	  "dbtags_Sterowanie".Zbiorniki_Godziny.Stop_napełnianie.HOUR := "dbHoldRegSlave_to_MT101".instHourStop_Filling;
	  "dbtags_Sterowanie".Zbiorniki_Godziny.Stop_napełnianie.MINUTE := "dbHoldRegSlave_to_MT101".instMinutStopt_Filling;
	  "dbtags_Sterowanie".Zbiorniki_Godziny.Stop_napełnianie.SECOND := 0;
	  
	  "dbtags_Sterowanie".Zbiorniki_Godziny.Start_przetłaczanie_1.HOUR := "dbHoldRegSlave_to_MT101".instHourStart_City;
	  "dbtags_Sterowanie".Zbiorniki_Godziny.Start_przetłaczanie_1.MINUTE := "dbHoldRegSlave_to_MT101".instMinutStart_City;
	  "dbtags_Sterowanie".Zbiorniki_Godziny.Start_przetłaczanie_1.SECOND := 0;
	  
	  "dbtags_Sterowanie".Zbiorniki_Godziny.Stop_przetłaczanie_1.HOUR := "dbHoldRegSlave_to_MT101".instHourStop_City;
	  "dbtags_Sterowanie".Zbiorniki_Godziny.Stop_przetłaczanie_1.MINUTE := "dbHoldRegSlave_to_MT101".instMinutStopt_City;
	  "dbtags_Sterowanie".Zbiorniki_Godziny.Stop_przetłaczanie_1.SECOND := 0;
	  
	  "dbtags_Sterowanie".Zbiorniki_Godziny.Start_dosilanie_1.HOUR := "dbHoldRegSlave_to_MT101".instHourStart_Replen;
	  "dbtags_Sterowanie".Zbiorniki_Godziny.Start_dosilanie_1.MINUTE := "dbHoldRegSlave_to_MT101".instMinutStart_Replen;
	  "dbtags_Sterowanie".Zbiorniki_Godziny.Start_dosilanie_1.SECOND := 0;
	  
	  "dbtags_Sterowanie".Zbiorniki_Godziny.Stop_dosilanie_1.HOUR := "dbHoldRegSlave_to_MT101".instHourStop_Replen;
	  "dbtags_Sterowanie".Zbiorniki_Godziny.Stop_dosilanie_1.MINUTE := "dbHoldRegSlave_to_MT101".instMinutStopt_Replen;
	  "dbtags_Sterowanie".Zbiorniki_Godziny.Stop_dosilanie_1.SECOND := 0;
	  
	  
	  
	  
	END_REGION
	
	
	
END_FUNCTION_BLOCK

FUNCTION "Zmienne_SCADA" : Void
{ S7_Optimized_Access := 'TRUE' }
VERSION : 0.1
   VAR_TEMP 
      TimeHz_DInt : DInt;
      TimeK1_ONDInt : DInt;
      TimeK2_ONDInt : DInt;
      TimeK1_OFFDInt : DInt;
      TimeK2_OFFDInt : DInt;
      tmpTimerSet_O2_Up : DInt;   // Pomocnicza wynik po mnozeniu [ms] czasu do zwiekszenia bar
      tmpQ1 : Int;   // pompcnicza przy konwersji z real do int
      tmpQ2 : Int;   // pompcnicza przy konwersji z real do int
   END_VAR


BEGIN
	(*
	//=============================================================================
	//(JZWiK S.A Radosław Tecmer)
	//(c)Copyright (2021) All Rights Reserved
	//-----------------------------------------------------------------------------
	//Testowane z:   (system docelowy z  FW 4.2)
	//Pakiet inżynierski:   TIA Portal (V14 Sp1 Update 9)
	//Ograniczenia:  ( - )
	//Wymagania:  (minimalne S7-1200 CPU 1214 FW 3.2 .)
	//Funkcjonalnośc: (Kopiowanie bloków danych z - do bloku SCADA )
	//-----------------------------------------------------------------------------
	//Zmainy wprowadzone:
	//Wersja  Data       Osoba wprowadzająca zmiany - ekspert
	//01.00.00 17.11.2021 (Tecmer Radosław - twórca) Pieresza wersja 01.00.00
	//=============================================================================
	*)
	
	//
	// Staus napędów P1 P2 P3 P4 POSTÓJ, FALOWNIK, SIEĆ
	//P1
	REGION Status napędów
	IF "IsRunInverter_P1" THEN
	  // Przekazanie wartości do instancji DB10 (1= falownik)
	  "db10organizacyjna".ins_ModeWorkContactronP1 := 1;
	  ;
	END_IF;
	IF "IsRunNetwork_P1" THEN
	  // Przekazanie wartości do instancji DB10 (2= sieć)
	  "db10organizacyjna".ins_ModeWorkContactronP1 := 2;
	  ;
	END_IF;
	IF ("IsRunNetwork_P1" = FALSE) AND ("IsRunInverter_P1" = FALSE) THEN
	  // Przekazanie wartości do instancji DB10 (0= postój)
	  "db10organizacyjna".ins_ModeWorkContactronP1 := 0;
	  ;
	END_IF;
	// P2
	IF "IsRunInverter_P2" THEN
	  // Przekazanie wartości do instancji DB10 (1= falownik)
	  "db10organizacyjna".ins_ModeWorkContactronP2 := 1;
	  ;
	END_IF;
	IF "IsRunNetwork_P2" THEN
	  // Przekazanie wartości do instancji DB10 (2= sieć)
	  "db10organizacyjna".ins_ModeWorkContactronP2 := 2;
	  ;
	END_IF;
	IF ("IsRunNetwork_P2" = FALSE) AND ("IsRunInverter_P2" = FALSE) THEN
	  // Przekazanie wartości do instancji DB10 (0= postój)
	  "db10organizacyjna".ins_ModeWorkContactronP2 := 0;
	  ;
	END_IF;
	//P3
	IF "IsRunInverter_P3" THEN
	  // Przekazanie wartości do instancji DB10 (1= falownik)
	  "db10organizacyjna".ins_ModeWorkContactronP3 := 1;
	  ;
	END_IF;
	IF "IsRunNetwork_P3" THEN
	  // Przekazanie wartości do instancji DB10 (2= sieć)
	  "db10organizacyjna".ins_ModeWorkContactronP3 := 2;
	  ;
	END_IF;
	IF ("IsRunNetwork_P3" = FALSE) AND ("IsRunInverter_P3" = FALSE) THEN
	  // Przekazanie wartości do instancji DB10 (0= postój)
	  "db10organizacyjna".ins_ModeWorkContactronP3 := 0;
	  ;
	END_IF;
	
	//P4
	IF "IsRunInverter_P4" THEN
	  // Przekazanie wartości do instancji DB10 (1= falownik)
	  "db10organizacyjna".ins_ModeWorkContactronP4 := 1;
	  ;
	END_IF;
	IF "IsRunNetwork_P4" THEN
	  // Przekazanie wartości do instancji DB10 (2= sieć)
	  "db10organizacyjna".ins_ModeWorkContactronP4 := 2;
	  ;
	END_IF;
	IF ("IsRunNetwork_P4" = FALSE) AND ("IsRunInverter_P4" = FALSE) THEN
	  // Przekazanie wartości do instancji DB10 (0= postój)
	  "db10organizacyjna".ins_ModeWorkContactronP4 := 0;
	  ;
	END_IF;
	
	//Zmienne na potrzreby trendów WinCC - Praca pomp
	//pompa P1
	IF ("IsRun_P1") = TRUE
	  
	THEN
	  "db10organizacyjna".act_stanP1 := 5;
	ELSE
	  "db10organizacyjna".act_stanP1 := 0;
	END_IF;
	//pompa P2
	IF ("IsRun_P2") = TRUE
	  
	THEN
	  "db10organizacyjna".act_statnP2 := 6;
	ELSE
	  "db10organizacyjna".act_statnP2 := 0;
	END_IF;
	//pompa P3
	IF ("IsRun_P3") = TRUE
	  
	THEN
	  "db10organizacyjna".act_stanP3 := 7;
	ELSE
	  "db10organizacyjna".act_stanP3 := 0;
	END_IF;
	
	//pompa P4
	IF ("IsRun_P3") = TRUE
	  
	THEN
	  "db10organizacyjna".act_stanP4 := 9;
	ELSE
	  "db10organizacyjna".act_stanP4 := 0;
	END_IF;
	
	
	// Zasuwy Pompownia
	// 
	// Status napędów Z11, 
	"dbdane".Z11_Status := "dbHoldRegSlave_to_MT101".instvValveZ11;
	// Status napędów Z12, 
	"dbdane".Z12_Status := "dbHoldRegSlave_to_MT101".instvValveZ12;
	
	// Staus napędów Z11 Z12
	"dbtags_Sterowanie".SetupControlPompownia.Z11_Status := "dbdane".Z11_Status;
	"dbtags_Sterowanie".SetupControlPompownia.Z12_Status := "dbdane".Z12_Status;
	
	END_REGION
	
	
	//********************
	
	
	REGION Region PID Zmienne
	  // Zmienne PID
	  //Limit górny wartości procesowej MV [%]
	  "dbdane"."PID_Compact_1_sPid_Cmpt.r_Lmn_Hlm" := "dbtags_Sterowanie".SetupControlPompownia.r_Lmn_Hlm;
	  "PID_Compact_1".sPid_Cmpt.r_Lmn_Hlm := "dbdane"."PID_Compact_1_sPid_Cmpt.r_Lmn_Hlm";
	  //Limit dolny wartości procesowej MV [%]
	  "dbdane"."PID_Compact_1_sPid_Cmpt.r_Lmn_Llm" := "dbtags_Sterowanie".SetupControlPompownia.r_Lmn_Llm;
	  "PID_Compact_1".sPid_Cmpt.r_Lmn_Llm := "dbdane"."PID_Compact_1_sPid_Cmpt.r_Lmn_Llm";
	  //Obiekt zreczywisty***
	  // Max wartość procesowa 
	  "dbdane"."PID_Compact_1sPid_Cmpt.r_Pv_Norm_OUT_2" := "dbtags_Sterowanie".SetupControlPompownia.r_Pv_Norm_OUT_2;
	  "PID_Compact_1".sPid_Cmpt.r_Pv_Norm_OUT_2 := "dbdane"."PID_Compact_1sPid_Cmpt.r_Pv_Norm_OUT_2";
	  //Min wartość procesowa
	  "dbdane"."PID_Compact_1_sPid_Cmpt.r_Pv_Norm_OUT_1" := "dbtags_Sterowanie".SetupControlPompownia.r_Pv_Norm_OUT_1;
	  "PID_Compact_1".sPid_Cmpt.r_Pv_Norm_OUT_1 := "dbdane"."PID_Compact_1_sPid_Cmpt.r_Pv_Norm_OUT_1";
	  //******
	  
	  
	  //Limmit górny zadawania
	  "dbdane"."PID_Compact_1_sPid_Cmpt.r_Sp_Hlm" := "dbtags_Sterowanie".SetupControlPompownia.r_Sp_Hlm;
	  "PID_Compact_1".sPid_Cmpt.r_Sp_Hlm := "dbdane"."PID_Compact_1_sPid_Cmpt.r_Sp_Hlm";
	  //Limit dolny zadawania
	  "dbdane"."PID_Compact_1_sPid_Cmpt.r_Sp_Llm" := "dbtags_Sterowanie".SetupControlPompownia.r_Sp_Llm;
	  "PID_Compact_1".sPid_Cmpt.r_Sp_Llm := "dbdane"."PID_Compact_1_sPid_Cmpt.r_Sp_Llm";
	  
	  // Setpoint SV
	  "db10organizacyjna".setpoint_SV_bar := "dbdane".Setpoint_SV;
	  
	END_REGION
	
	REGION Sterowanie czasem zmiany wartości ciśnienia w modelu regulacji nadążnej 
	  
	  //Opóznienie zwiększania watrości ciśnieniea  konwersja i przekaznie do zmiennej tymczasowej 
	  #tmpTimerSet_O2_Up := INT_TO_DINT("db10organizacyjna".TimeHistere_set_bar);
	  
	  //Przekazanie do Timera -Zadany czas [ms] zwłoki zwiekszenia ciśnienia
	  "dbtags_Sterowanie".SetupControlPompownia.TimerSet_O2_Up.PT := DINT_TO_TIME(#tmpTimerSet_O2_Up * "MS_TO_M");
	  //Przekazanie do Timera -Zadany czas [ms] zwłoki zmniejszenia ciśnienie
	  "dbtags_Sterowanie".SetupControlPompownia.TimerSet_O2_Down.PT := DINT_TO_TIME(#tmpTimerSet_O2_Up * "MS_TO_M");
	  
	END_REGION
	
	REGION Timery dołączenia dodatkowych pomp 
	  //***Czasy dołącz wyłacz pompy dodatkowa i oczekiwanie na Hz50 ***//
	  
	  "dbtags_Sterowanie".SetupControlPompownia.Time_ONK1 := "db10organizacyjna".Time_ONK1;
	  "dbtags_Sterowanie".SetupControlPompownia.Time_ONK2 := "db10organizacyjna".Time_ONK2;
	  "dbtags_Sterowanie".SetupControlPompownia.Time_OFFK1 := "db10organizacyjna".Time_OFFK1;
	  "dbtags_Sterowanie".SetupControlPompownia.Time_OFFK2 := "db10organizacyjna".Time_OFFK2;
	  "dbtags_Sterowanie".SetupControlPompownia.TimeHz := "db10organizacyjna".TimeHz;
	  
	  
	END_REGION
	
	
	//**
	"dbtags_Sterowanie".SetupControlPompownia.tagsdbSwitch_ModelSterowania := "dbdane".Switch_model_control_P1P4;
	
	
	
	REGION Przekazanie zmiennych sterowania
	  
	  //Wspólczynnik korekty ostrzeżęń wyokiego i niskiego PV HWrn, PV LWrn 
	  //Wsółcynnik ten koryguje poziom alarmu PID górnego i dolnego odpowiadających
	  //za dołączenie i odączenie dodatkowych kompresorów 
	  "dbtags_Sterowanie".SetupControlPompownia.PV_HWrn_correction := "db10organizacyjna".PV_HWrn_set_correct;
	  "dbtags_Sterowanie".SetupControlPompownia.PV_LWrn_correction := "db10organizacyjna".PV_LWrn_set_correct;
	  
	  //Czas oczekiwania na 50 Hz  konwersja i przekaznie do zmiennej tymczasowej 
	  #TimeHz_DInt := INT_TO_DINT("db10organizacyjna".TimeHz);
	  
	  //Czas oczekiwania na 50Hz 
	  "dbdane".TMR_Hz := DINT_TO_TIME(#TimeHz_DInt * "MS_TO_S");
	  
	  //Czas oczekiwania na K1_ON  konwersja i przekaznie do zmiennej tymczasowej 
	  #TimeK1_ONDInt := INT_TO_DINT("db10organizacyjna".Time_ONK1);
	  
	  //Czas oczekiwania na K1_ON 
	  "dbdane".TMR_ON_K1 := DINT_TO_TIME(#TimeK1_ONDInt * "MS_TO_S");
	  
	  //Czas oczekiwania na K1_OFF  konwersja i przekaznie do zmiennej tymczasowej 
	  #TimeK1_OFFDInt := INT_TO_DINT("db10organizacyjna".Time_OFFK1);
	  
	  //Czas oczekiwania na K1_OFF 
	  "dbdane".TMR_OFF_K1 := DINT_TO_TIME(#TimeK1_OFFDInt * "MS_TO_S");
	  
	  //Czas oczekiwania na K2_ON  konwersja i przekaznie do zmiennej tymczasowej 
	  #TimeK2_ONDInt := INT_TO_DINT("db10organizacyjna".Time_ONK2);
	  
	  //Czas oczekiwania na K2_ON 
	  "dbdane".TMR_ON_K2 := DINT_TO_TIME(#TimeK2_ONDInt * "MS_TO_S");
	  
	  //Czas oczekiwania na K2_OFF  konwersja i przekaznie do zmiennej tymczasowej 
	  #TimeK2_OFFDInt := INT_TO_DINT("db10organizacyjna".Time_OFFK2);
	  
	  //Czas oczekiwania na K2_OFF 
	  "dbdane".TMR_OFF_K2 := DINT_TO_TIME(#TimeK2_OFFDInt * "MS_TO_S");
	  
	  //Aktualne Hz przekazane do instancji SCADA
	  "db10organizacyjna".set_Hz_P1P4 := "dbdane".OUT_PURE_Real;
	  
	  //Aktualna zadana wartość ciśnienia do regulatora
	  CASE "dbHoldRegSlave_to_MT101".instSygSter_1 OF
	    1:
	      "dbdane".Setpoint_SV := "dbHoldRegSlave_to_MT101".instSetbarDN500_B5;
	    2:
	      "dbdane".Setpoint_SV := "dbHoldRegSlave_to_MT101".instSetbarDN225_B6;
	    3:
	      "dbdane".Setpoint_SV := "dbdane".Setpoint_bar_automat;
	      
	    ELSE
	      "dbdane".Setpoint_SV := 0.0;
	      ;
	  END_CASE;
	  
	END_REGION
	
	
	REGION Analogi 
	  
	//************ parametry analogowe**************
	//Przekazane z PLC - Zasuwy
	  "dbdane".Act_Value_B5_magistrala_bar := "dbHold_RRG".actB5_bar_magistrala;
	
	//Aktualna mierzona wartość ciśnienia zasilania B5
	"db10organizacyjna".instB5_bar_act_magistrala := "dbdane".Act_Value_B5_magistrala_bar;
	
	//Aktualna mierzona wartość ciśnienia  kierunek miasto B6
	"db10organizacyjna".instB6_bar_act_miasto := "dbdane".act_Value_B6;
	
	//Aktualna mierzona wartość ciśnienia  pompownia B7
	"db10organizacyjna".instB7_bar_act_pompownia := "dbdane".act_Value_B7;
	
	//Aktualna średnia wyliczona wartość ciśnienia 
	//Wyliczanie następuje dopiero po wybraniu sterowania od wartości średniej
	"db10organizacyjna".avg_bar:= "dbdane".actPrzepływQ1_IA_real;
	
	// Aktualne ciśnienie suchobiegu
	"db10organizacyjna".instB8_bar_act_suchobieg := "dbdane".act_Value_B8;
	END_REGION
	
	//Przekazanie zmiennej tryb pracy PID - SYMULACJA TESTY
	//IF "Sumul_OnOFF_manual_PID" = FALSE THEN
	  // ustaw trzb PID na automat
	//  "PID_Compact_1".sRet.i_Mode := "dbtags_Sterowanie".PID_Compact.Mode;
	//  ;
	//END_IF;
	
	
	REGION Alarmy 
	  // Sygnały alarmów systemu sterowania i komunikacji
	  "HMI.alarm_02" := "dbzarządzanie".sterowanie_1."alarm-warning";
	  "HMI.alarm_01" := "dbzarządzanie".sterowanie_1."alarm-modbus";
	  
	  
	END_REGION
	
	
	//Przekazanie bitu kasowania Alarmu PIEZO
	//...........
	
	
	// Falownik i zasilania RS
	REGION Counter Event OverTemp's OverVolt's from Inverters
	  // Falownik pomp
	  "db10organizacyjna".CounterOverTempFa := "dbMasterData".data26_Inver_OverTemp_415040_Fal.typeDataInverter_int[0];
	  "db10organizacyjna".CounterOverVoltFal := "dbMasterData".data26_Inver_OverVolts_415050_Fal.typeDataInverter_int[0];
	  "HMI.gotowość_falownik_1" := "dbzarządzanie".awaria_falownika_F1;
	  // RS
	  "HMI.brak_zasilania" := "dbzarządzanie".brak_zasilania_RS;
	  
	
	END_REGION
	
	
	REGION Manual zadane Hz (SV)
	  // konwertowanie wartości manualnie zadawanych Hz z Real do Word
	  "dbdane".tmpManualSV := REAL_TO_LREAL("dbdane".Manual_SV);
	  "dbdane".ManualSV_Int := LREAL_TO_INT( "dbdane".tmpManualSV);
	 
	  
	END_REGION
	
	
	
	REGION Modbus staus, error
	  // Status Modbus slave
	  "db10organizacyjna".RTU_MPP04_1errorStatus := "dbTags_master_MPP04_1".modbusMaster.errorStatus;
	  "db10organizacyjna".RTU_MPP04_2errorStatus := "dbTags_master_MPP04_2".modbusMaster.errorStatus;
	  "db10organizacyjna".RTU_Fal_1errorStatus := "dbTags_master_Fal_1".modbusMaster.errorStatus;
	  //Status Modbus master
	  "db10organizacyjna".RTU_MT101 := "dbTags_slave_RTU".modbusMaster.errorStatus;
	  %DB10.DBX25.0 := "dbzarządzanie".sterowanie_1.awaria_modbus_falownik;
	  %DB10.DBX25.1 := "dbzarządzanie".sterowanie_1.awaria_modbus_przepływ_pomp;
	  %DB10.DBX25.2 := "dbzarządzanie".sterowanie_1.awaria_modbus_przepływ_magist;
	  %DB10.DBX25.3 := "dbzarządzanie".sterowanie_1.awaria_modbus_mt101;
	  
	  
	END_REGION
	
	REGION Modbus master PLC S7 1200 - Przepływomierz Q1 pompownia
	  // przekazanie wartości Real
	  "db10organizacyjna".instFlowDN225_act_Q1 := "dbdane".Wielkość_przeływu_Q1;
	  
	  // konwertowanie do Int
	  "db10organizacyjna".actQ1_przepyw_pompownia_Int := "dbdane".actPrzeoływQ1;
	  
	  // Sumay przepływu 
	  "db10organizacyjna".instSumFlowDN225_Q1 := "dbdane".Licznik_objętość_VF_Q1;
	  
	  
	  //******* Dopisać jeśli potzrebne do wizualizacji 
	  // Adres 2 - Licznik_objętość_VF
	  // Adres 4- stan bierzący licznika objetości w stecz VR
	  // Adres 6- stan bierzący licznika różnicowego  objętości VD
	  // Adres 8- główny liczni objetości w przód GF
	  // Adres 10- główny liczni objetości w stecz GR
	  // Adres 12- główny lróznicowy liczni objetościGD
	  // Status MP04 Q1 - pompownia
	  
	  
	END_REGION
	
	
	REGION Modbus master PLC S7 1200 - Przepływomierz Q2 Zasuwy
	  // przekazanie wartości
	  "db10organizacyjna".instFlowDN500_act_Q2 := "dbdane".Wielkość_przeływu_Q2;
	  
	  // konwertowanie do Int
	  #tmpQ2 := REAL_TO_INT("db10organizacyjna".instFlowDN500_act_Q2);
	  "db10organizacyjna".actQ2_przepyw_pompownia_Int := #tmpQ2;
	  
	  //******* Dopisać jeśli potzrebne do wizualizacji 
	  // Adres 2 - Licznik_objętość_VF
	  // Adres 4- stan bierzący licznika objetości w stecz VR
	  // Adres 6- stan bierzący licznika różnicowego  objętości VD
	  // Adres 8- główny liczni objetości w przód GF
	  // Adres 10- główny liczni objetości w stecz GR
	  // Adres 12- główny lróznicowy liczni objetościGD
	  // Status MP04 Q1 - pompownia
	  
	  
	  
	  // Sumay przepływu 
	  "db10organizacyjna".instSumFlowDN500_Q2 := "dbdane".Licznik_objętość_VF_Q2;
	  
	END_REGION
	
	REGION Modbus RTU Falownik 
	  // Słowo statusu 
	  "HMI.SłowoStatus_Falownik1" := "dbModbusRTU_Reg".received26_Inver_Status_word_416030.typeDataInverter_int[0];
	  
	END_REGION
	
	REGION położenie Z10
	  // kopiowanie odebranych danych z PLC Zasuwy
	  "dbHoldRegSlave_to_MT101".instPozitionZ10_act := INT_TO_REAL("db10organizacyjna".actPozycja_Z10);
	  
	END_REGION
	
	
	
	
	
	
	  
	  
	
	
	
	
END_FUNCTION

FUNCTION "Konwersja_Time_to_Int" : Void
{ S7_Optimized_Access := 'TRUE' }
AUTHOR : RTecmer
FAMILY : 'HMI(XM)'
VERSION : 0.1
//Przekazywanie zmiennych między urządzeniami

BEGIN
	(*
	//=============================================================================
	//(JZWiK S.A Radosław Tecmer)
	//(c)Copyright (2021) All Rights Reserved
	//-----------------------------------------------------------------------------
	//Testowane z:   (system docelowy z  FW 4.2)
	//Pakiet inżynierski:   TIA Portal (V14 Sp1 Update 9)
	//Ograniczenia:  ( - )
	//Wymagania:  (minimalne S7-1200 CPU 1214 FW 3.2 .)
	//Funkcjonalnośc: (KOnwerja zmiennych formatu Time of Day na Int )
	//-----------------------------------------------------------------------------
	//Zmainy wprowadzone:
	//Wersja  Data       Osoba wprowadzająca zmiany - ekspert
	//01.00.00 17.02.2022 (Tecmer Radosław - twórca) Pieresza wersja 01.00.00
	//=============================================================================
	*)
	
	// Aktualny czas
	"Konverter_zegarów"(HOUR:="Data_Czas_synch".Time_Local_read.HOUR,
	                    MINUTE:="Data_Czas_synch".Time_Local_read.MINUTE,
	                    SECOND:="Data_Czas_synch".Time_Local_read.SECOND,
	                    Czas_Liczba_conv_Real=>"db10organizacyjna".actTime,
	                    Zegar_H=>"db10organizacyjna".actHour,
	                    Zegar_M=>"db10organizacyjna".actMinut,
	                    Zegar_S=>"db10organizacyjna".actSec);
	
	
	// Godzina start napełniania
	"Konverter_zegarów"(HOUR:="db10organizacyjna".instHourStart_Filling.HOUR,
	                    MINUTE:="db10organizacyjna".instHourStart_Filling.MINUTE,
	                    SECOND:="db10organizacyjna".instHourStart_Filling.SECOND,
	                    Czas_Liczba_conv_Real=>"dbzarządzanie".instHourStart_Filling,
	                    Zegar_H=>"db10organizacyjna".instHourStart_Filling_1,
	                    Zegar_M=>"db10organizacyjna".instMinutStart_Filling,
	                    Zegar_S=>"db10organizacyjna".instSecStart_Filling_1);
	
	
	// Godzina stop napełniania
	"Konverter_zegarów"(HOUR := "db10organizacyjna".instHourStop_Filling.HOUR,
	                    MINUTE := "db10organizacyjna".instHourStop_Filling.MINUTE,
	                    SECOND := "db10organizacyjna".instHourStop_Filling.SECOND,
	                    Czas_Liczba_conv_Real => "dbzarządzanie".instHourStop_Filling,
	                    Zegar_H=>"db10organizacyjna".instHourStop_Filling_1,
	                    Zegar_M=>"db10organizacyjna".instMinutStopt_Filling,
	                    Zegar_S=>"db10organizacyjna".instSecStop_Filling_1);
	
	// Godzina start przetłaczanie miasto DN225
	"Konverter_zegarów"(HOUR := "db10organizacyjna".instHourStart_City.HOUR,
	                    MINUTE := "db10organizacyjna".instHourStart_City.MINUTE,
	                    SECOND := "db10organizacyjna".instHourStart_City.SECOND,
	                    Czas_Liczba_conv_Real => "dbzarządzanie".instHourStart_City,
	                    Zegar_H=>"db10organizacyjna".instHourStart_City_1,
	                    Zegar_M=>"db10organizacyjna".instMinutStart_City,
	                    Zegar_S=>"db10organizacyjna".instSecStart_City_1);
	
	
	// Godzina stop przetłaczanie miasto DN225
	"Konverter_zegarów"(HOUR := "db10organizacyjna".instHourStop_City.HOUR,
	                    MINUTE := "db10organizacyjna".instHourStop_City.MINUTE,
	                    SECOND := "db10organizacyjna".instHourStop_City.SECOND,
	                    Czas_Liczba_conv_Real => "dbzarządzanie".instHourStop_City,
	                    Zegar_H=>"db10organizacyjna".instHourStop_City_1,
	                    Zegar_M=>"db10organizacyjna".instMinutStopt_City,
	                    Zegar_S=>"db10organizacyjna".instSecStop_City_1);
	
	
	// Godzina start dosilanie DN500
	"Konverter_zegarów"(HOUR := "db10organizacyjna".instHourStart_Replen.HOUR,
	                    MINUTE := "db10organizacyjna".instHourStart_Replen.MINUTE,
	                    SECOND := "db10organizacyjna".instHourStart_Replen.SECOND,
	                    Czas_Liczba_conv_Real => "dbzarządzanie".instHourStart_Replen,
	                    Zegar_H=>"db10organizacyjna".instHourStart_Replen_1,
	                    Zegar_M=>"db10organizacyjna".instMinutStart_Replen,
	                    Zegar_S=>"db10organizacyjna".instSecStart_Replen_1);
	
	
	
	
	
	// Godzina stop dosilanie DN500
	"Konverter_zegarów"(HOUR :="db10organizacyjna".instHourStop_Replen.HOUR,
	                    MINUTE :="db10organizacyjna".instHourStop_Replen.MINUTE,
	                    SECOND :="db10organizacyjna".instHourStop_Replen.SECOND,
	                    Czas_Liczba_conv_Real => "dbzarządzanie".instHourStop_Replen,
	                    Zegar_H=>"db10organizacyjna".instHourStop_Replen_1,
	                    Zegar_M=>"db10organizacyjna".instMinutStopt_Replen,
	                    Zegar_S=>"db10organizacyjna".instSecStop_Replen_1);
	
	
	
	
	
	
	
	
	
	
	
END_FUNCTION

FUNCTION "Konverter_zegarów" : Void   // FC31, LAD
{ S7_Optimized_Access := 'FALSE' }
VERSION : 0.1
// stored: AutoNumber true, IsIECCheckEnabled false, SetENOAutomatically false, UDAEnableTagReadback false
   VAR_INPUT
      HOUR : USInt;   // Zmienna godzina z DTL
      MINUTE : USInt;   // Zmienna minuty z DTL
      SECOND : USInt;   // Zmienne sekundy z DTL
   END_VAR
   VAR_OUTPUT
      Czas_Liczba_conv_Real : Real;   // Liczba przedstawiająca czas 00:00:00 liczbowo 00.0000
      Zegar_H : Int;
      Zegar_M : Int;
      Zegar_S : Int;
   END_VAR
   VAR_TEMP
      zegar_H_pomocnicza : Real;   // pomocnicza do przekształcenia czasu z DLT do Real
      zegar_M_pomocnicza : Real;   // pomocnicza do przekształcenia czasu z DLT do Real
      zegar_S_pomocnicza : Real;   // pomocnicza do przekształcenia czasu z DLT do Real
      zegar_H_Uint : UInt;   // pomocnicza do przekształcenia czasu z DLT do Uint
      zegar_M_Uint : UInt;   // pomocnicza do przekształcenia czasu z DLT do Uint
      zegar_S_Uint : UInt;   // pomocnicza do przekształcenia czasu z DLT do Uint
   END_VAR
BEGIN

REGION Network 1: Wyodrębnienie zegara z danej DTL czasu lokalnego
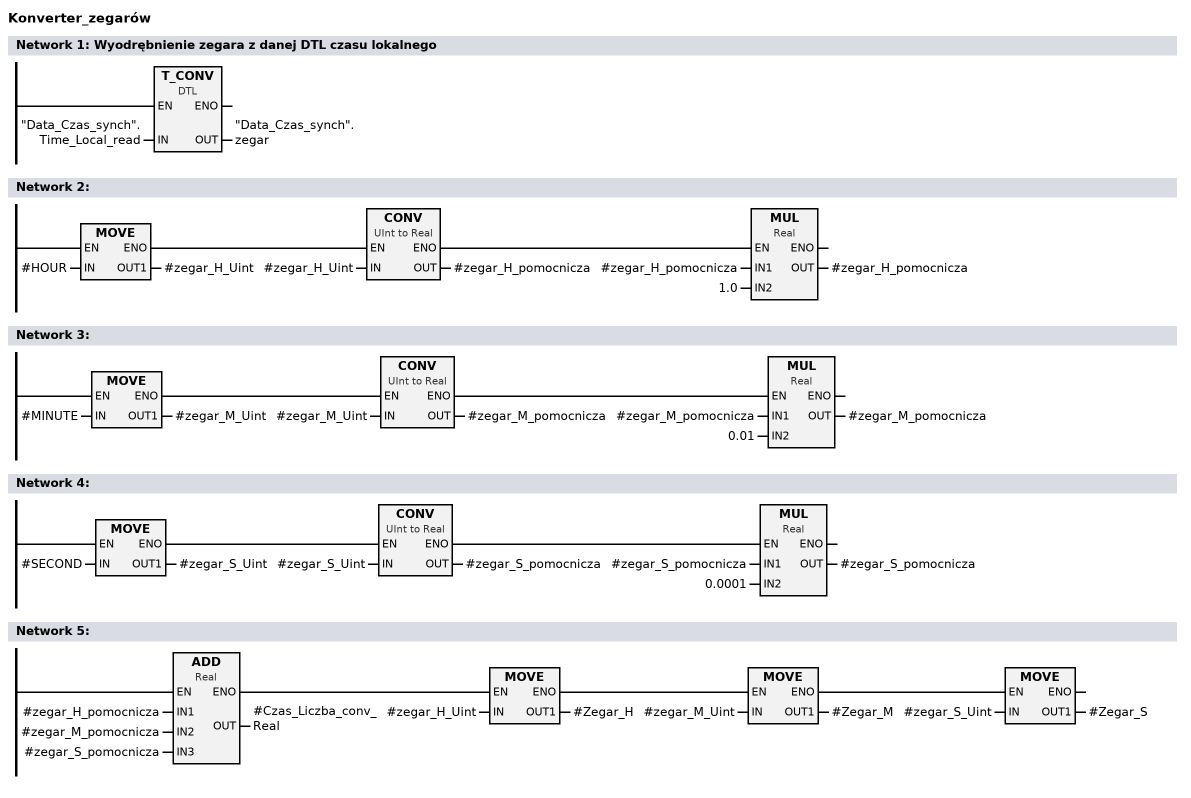
   RUNG wire#powerrail
      { S7_Templates := "[src_type := DTL, dest_type := Time_Of_Day]" } T_CONV(IN := "Data_Czas_synch".Time_Local_read, OUT => "Data_Czas_synch".zegar)
   END_RUNG
   // the same network as SCL:
   T_CONV(IN := "Data_Czas_synch".Time_Local_read, OUT => "Data_Czas_synch".zegar);
END_REGION

REGION Network 2
   RUNG wire#powerrail
      { S7_GenerateENO := "TRUE" } Move(in := #HOUR, out1 => #zegar_H_Uint)
      { S7_Templates := "[SrcType := UInt, DestType := Real]"; S7_GenerateENO := "TRUE" } Convert(in := #zegar_H_Uint, out => #zegar_H_pomocnicza)
      { S7_Templates := "SrcType := Real"; S7_GenerateENO := "TRUE" } Mul(in1 := #zegar_H_pomocnicza, in2 := 1.0, out => #zegar_H_pomocnicza)
   END_RUNG
   // the same network as SCL:
   // ENO of a box is taken as its EN; it also drops when the box reports an error
   #zegar_H_Uint := #HOUR;
   #zegar_H_pomocnicza := UINT_TO_REAL(#zegar_H_Uint);
   #zegar_H_pomocnicza := #zegar_H_pomocnicza * 1.0;
END_REGION

REGION Network 3
   RUNG wire#powerrail
      { S7_GenerateENO := "TRUE" } Move(in := #MINUTE, out1 => #zegar_M_Uint)
      { S7_Templates := "[SrcType := UInt, DestType := Real]"; S7_GenerateENO := "TRUE" } Convert(in := #zegar_M_Uint, out => #zegar_M_pomocnicza)
      { S7_Templates := "SrcType := Real"; S7_GenerateENO := "TRUE" } Mul(in1 := #zegar_M_pomocnicza, in2 := 0.01, out => #zegar_M_pomocnicza)
   END_RUNG
   // the same network as SCL:
   // ENO of a box is taken as its EN; it also drops when the box reports an error
   #zegar_M_Uint := #MINUTE;
   #zegar_M_pomocnicza := UINT_TO_REAL(#zegar_M_Uint);
   #zegar_M_pomocnicza := #zegar_M_pomocnicza * 0.01;
END_REGION

REGION Network 4
   RUNG wire#powerrail
      { S7_GenerateENO := "TRUE" } Move(in := #SECOND, out1 => #zegar_S_Uint)
      { S7_Templates := "[SrcType := UInt, DestType := Real]"; S7_GenerateENO := "TRUE" } Convert(in := #zegar_S_Uint, out => #zegar_S_pomocnicza)
      { S7_Templates := "SrcType := Real"; S7_GenerateENO := "TRUE" } Mul(in1 := #zegar_S_pomocnicza, in2 := 0.0001, out => #zegar_S_pomocnicza)
   END_RUNG
   // the same network as SCL:
   // ENO of a box is taken as its EN; it also drops when the box reports an error
   #zegar_S_Uint := #SECOND;
   #zegar_S_pomocnicza := UINT_TO_REAL(#zegar_S_Uint);
   #zegar_S_pomocnicza := #zegar_S_pomocnicza * 0.0001;
END_REGION

REGION Network 5
   RUNG wire#powerrail
      { S7_Templates := "SrcType := Real"; S7_GenerateENO := "TRUE" } Add(in1 := #zegar_H_pomocnicza, in2 := #zegar_M_pomocnicza, in3 := #zegar_S_pomocnicza, out => #Czas_Liczba_conv_Real)
      Move(in := #zegar_H_Uint, out1 => #Zegar_H)
      Move(in := #zegar_M_Uint, out1 => #Zegar_M)
      Move(in := #zegar_S_Uint, out1 => #Zegar_S)
   END_RUNG
   // the same network as SCL:
   // ENO of a box is taken as its EN; it also drops when the box reports an error
   #Czas_Liczba_conv_Real := #zegar_H_pomocnicza + #zegar_M_pomocnicza + #zegar_S_pomocnicza;
   #Zegar_H := #zegar_H_Uint;
   #Zegar_M := #zegar_M_Uint;
   #Zegar_S := #zegar_S_Uint;
END_REGION
END_FUNCTION

FUNCTION "Kontrola trybu sterowania" : Void   // FC27, LAD
{ S7_Optimized_Access := 'TRUE' }
AUTHOR : rtecmer
VERSION : 0.1
// Kontrola trybu pracy Manual/Automat. Kontrola trybu pracy PID tryb 4 / tryb 3. Sprawdzanie stanu otwarcia Z11, Z12. Sprawdzanie sygnału Alarm Suchobieg. Tryb sterownia zostaje przerwany w wypadku wystąpienia 'Suchobiegu", lub zamknięcia obu zasów Z11 i Z12
// stored: AutoNumber true, IsIECCheckEnabled false, SetENOAutomatically false, UDAEnableTagReadback false
   VAR_IN_OUT
      Timer_Reset_delay : TOF_TIME;
   END_VAR
   VAR_TEMP   // added for the SCL form of the ladder/FBD networks
      _w1 : Bool;
      _w2 : Bool;
   END_VAR
BEGIN

REGION Network 1: Ustawienie pracy [Automat]
   // Ustawienie bitu [Automat] przełacznikiem trybu pracy
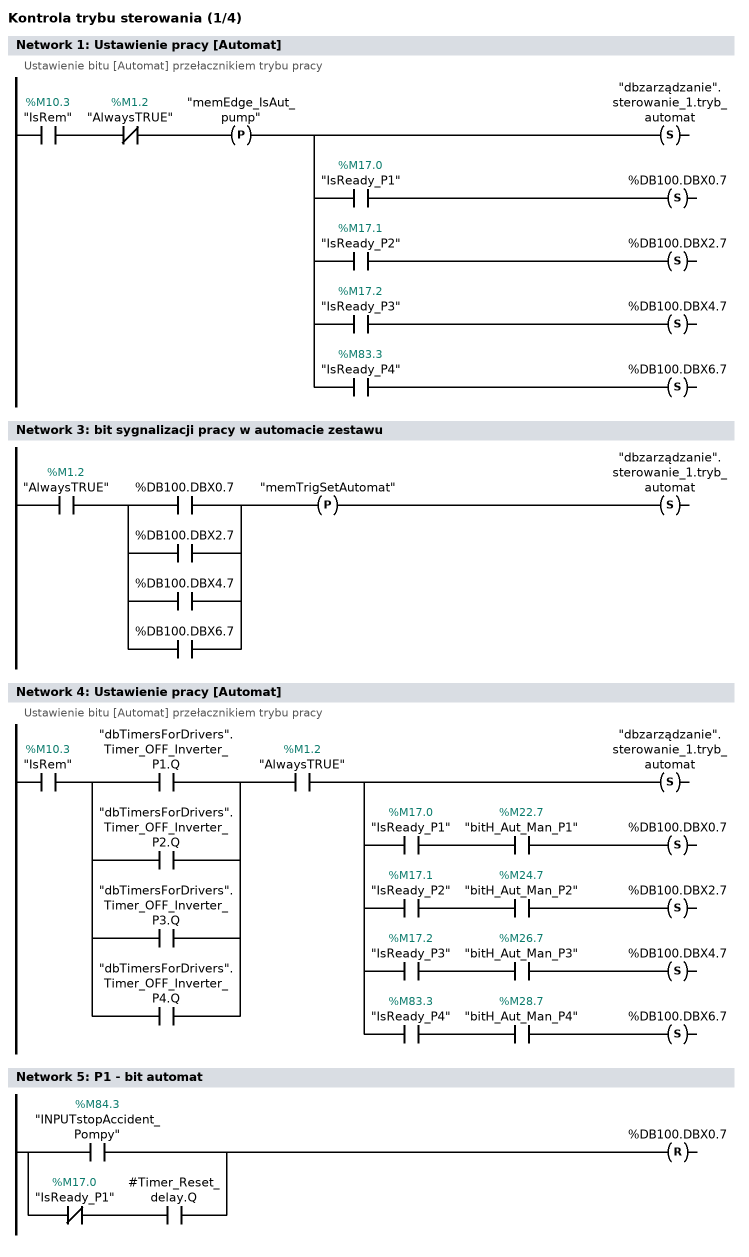
   RUNG wire#powerrail
      Contact( "IsRem" )
      I_Contact( "AlwaysTRUE" )
      P_Trig( "memEdge_IsAut_pump" )
      wire#w1
      S_Coil( "dbzarządzanie".sterowanie_1.tryb_automat )
   END_RUNG
   RUNG wire#w1
      Contact( "IsReady_P1" )
      S_Coil( %DB100.DBX0.7 )
   END_RUNG
   RUNG wire#w1
      Contact( "IsReady_P2" )
      S_Coil( %DB100.DBX2.7 )
   END_RUNG
   RUNG wire#w1
      Contact( "IsReady_P3" )
      S_Coil( %DB100.DBX4.7 )
   END_RUNG
   RUNG wire#w1
      Contact( "IsReady_P4" )
      S_Coil( %DB100.DBX6.7 )
   END_RUNG
   // the same network as SCL:
   #_w1 := "IsRem" AND NOT "AlwaysTRUE";
   #_w2 := #_w1 AND NOT "memEdge_IsAut_pump";   // rising edge
   "memEdge_IsAut_pump" := #_w1;
   IF #_w2 THEN "dbzarządzanie".sterowanie_1.tryb_automat := TRUE; END_IF;
   IF #_w2 AND "IsReady_P1" THEN %DB100.DBX0.7 := TRUE; END_IF;
   IF #_w2 AND "IsReady_P2" THEN %DB100.DBX2.7 := TRUE; END_IF;
   IF #_w2 AND "IsReady_P3" THEN %DB100.DBX4.7 := TRUE; END_IF;
   IF #_w2 AND "IsReady_P4" THEN %DB100.DBX6.7 := TRUE; END_IF;
END_REGION

REGION Network 3: bit sygnalizacji pracy w automacie zestawu
   RUNG wire#powerrail
      Contact( "AlwaysTRUE" )
      wire#w1
      Contact( %DB100.DBX0.7 )
      wire#w2
      P_Trig( "memTrigSetAutomat" )
      S_Coil( "dbzarządzanie".sterowanie_1.tryb_automat )
   END_RUNG
   RUNG wire#w1
      Contact( %DB100.DBX2.7 )
   END_RUNG wire#w2
   RUNG wire#w1
      Contact( %DB100.DBX4.7 )
   END_RUNG wire#w2
   RUNG wire#w1
      Contact( %DB100.DBX6.7 )
   END_RUNG wire#w2
   // the same network as SCL:
   #_w1 := "AlwaysTRUE" AND (%DB100.DBX0.7 OR %DB100.DBX2.7 OR %DB100.DBX4.7 OR %DB100.DBX6.7);
   #_w2 := #_w1 AND NOT "memTrigSetAutomat";   // rising edge
   "memTrigSetAutomat" := #_w1;
   IF #_w2 THEN "dbzarządzanie".sterowanie_1.tryb_automat := TRUE; END_IF;
END_REGION

REGION Network 4: Ustawienie pracy [Automat]
   // Ustawienie bitu [Automat] przełacznikiem trybu pracy
   RUNG wire#powerrail
      Contact( "IsRem" )
      wire#w1
      Contact( "dbTimersForDrivers".Timer_OFF_Inverter_P1.Q )
      wire#w2
      Contact( "AlwaysTRUE" )
      wire#w3
      S_Coil( "dbzarządzanie".sterowanie_1.tryb_automat )
   END_RUNG
   RUNG wire#w1
      Contact( "dbTimersForDrivers".Timer_OFF_Inverter_P2.Q )
   END_RUNG wire#w2
   RUNG wire#w1
      Contact( "dbTimersForDrivers".Timer_OFF_Inverter_P3.Q )
   END_RUNG wire#w2
   RUNG wire#w1
      Contact( "dbTimersForDrivers".Timer_OFF_Inverter_P4.Q )
   END_RUNG wire#w2
   RUNG wire#w3
      Contact( "IsReady_P1" )
      Contact( "bitH_Aut_Man_P1" )
      S_Coil( %DB100.DBX0.7 )
   END_RUNG
   RUNG wire#w3
      Contact( "IsReady_P2" )
      Contact( "bitH_Aut_Man_P2" )
      S_Coil( %DB100.DBX2.7 )
   END_RUNG
   RUNG wire#w3
      Contact( "IsReady_P3" )
      Contact( "bitH_Aut_Man_P3" )
      S_Coil( %DB100.DBX4.7 )
   END_RUNG
   RUNG wire#w3
      Contact( "IsReady_P4" )
      Contact( "bitH_Aut_Man_P4" )
      S_Coil( %DB100.DBX6.7 )
   END_RUNG
   // the same network as SCL:
   #_w1 := "IsRem" AND ("dbTimersForDrivers".Timer_OFF_Inverter_P1.Q OR "dbTimersForDrivers".Timer_OFF_Inverter_P2.Q OR "dbTimersForDrivers".Timer_OFF_Inverter_P3.Q OR "dbTimersForDrivers".Timer_OFF_Inverter_P4.Q) AND "AlwaysTRUE";
   IF #_w1 THEN "dbzarządzanie".sterowanie_1.tryb_automat := TRUE; END_IF;
   IF #_w1 AND "IsReady_P1" AND "bitH_Aut_Man_P1" THEN %DB100.DBX0.7 := TRUE; END_IF;
   IF #_w1 AND "IsReady_P2" AND "bitH_Aut_Man_P2" THEN %DB100.DBX2.7 := TRUE; END_IF;
   IF #_w1 AND "IsReady_P3" AND "bitH_Aut_Man_P3" THEN %DB100.DBX4.7 := TRUE; END_IF;
   IF #_w1 AND "IsReady_P4" AND "bitH_Aut_Man_P4" THEN %DB100.DBX6.7 := TRUE; END_IF;
END_REGION

REGION Network 5: P1 - bit automat
   RUNG wire#powerrail
      Contact( "INPUTstopAccident_Pompy" )
      wire#w1
      R_Coil( %DB100.DBX0.7 )
   END_RUNG
   RUNG wire#powerrail
      I_Contact( "IsReady_P1" )
      Contact( #Timer_Reset_delay.Q )
   END_RUNG wire#w1
   // the same network as SCL:
   IF "INPUTstopAccident_Pompy" OR (NOT "IsReady_P1" AND #Timer_Reset_delay.Q) THEN
       %DB100.DBX0.7 := FALSE;
   END_IF;
END_REGION

REGION Network 6: P2 - bit automat
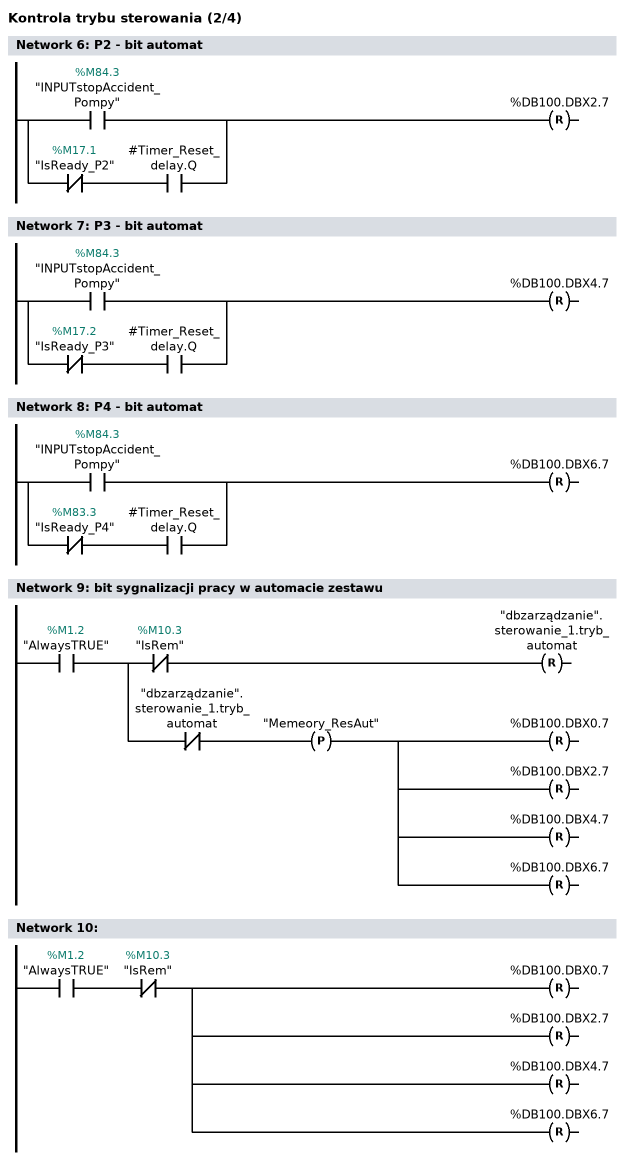
   RUNG wire#powerrail
      Contact( "INPUTstopAccident_Pompy" )
      wire#w1
      R_Coil( %DB100.DBX2.7 )
   END_RUNG
   RUNG wire#powerrail
      I_Contact( "IsReady_P2" )
      Contact( #Timer_Reset_delay.Q )
   END_RUNG wire#w1
   // the same network as SCL:
   IF "INPUTstopAccident_Pompy" OR (NOT "IsReady_P2" AND #Timer_Reset_delay.Q) THEN
       %DB100.DBX2.7 := FALSE;
   END_IF;
END_REGION

REGION Network 7: P3 - bit automat
   RUNG wire#powerrail
      Contact( "INPUTstopAccident_Pompy" )
      wire#w1
      R_Coil( %DB100.DBX4.7 )
   END_RUNG
   RUNG wire#powerrail
      I_Contact( "IsReady_P3" )
      Contact( #Timer_Reset_delay.Q )
   END_RUNG wire#w1
   // the same network as SCL:
   IF "INPUTstopAccident_Pompy" OR (NOT "IsReady_P3" AND #Timer_Reset_delay.Q) THEN
       %DB100.DBX4.7 := FALSE;
   END_IF;
END_REGION

REGION Network 8: P4 - bit automat
   RUNG wire#powerrail
      Contact( "INPUTstopAccident_Pompy" )
      wire#w1
      R_Coil( %DB100.DBX6.7 )
   END_RUNG
   RUNG wire#powerrail
      I_Contact( "IsReady_P4" )
      Contact( #Timer_Reset_delay.Q )
   END_RUNG wire#w1
   // the same network as SCL:
   IF "INPUTstopAccident_Pompy" OR (NOT "IsReady_P4" AND #Timer_Reset_delay.Q) THEN
       %DB100.DBX6.7 := FALSE;
   END_IF;
END_REGION

REGION Network 9: bit sygnalizacji pracy w automacie zestawu
   RUNG wire#powerrail
      Contact( "AlwaysTRUE" )
      wire#w1
      I_Contact( "IsRem" )
      R_Coil( "dbzarządzanie".sterowanie_1.tryb_automat )
   END_RUNG
   RUNG wire#w1
      I_Contact( "dbzarządzanie".sterowanie_1.tryb_automat )
      P_Trig( "Memeory_ResAut" )
      wire#w2
      R_Coil( %DB100.DBX0.7 )
   END_RUNG
   RUNG wire#w2
      R_Coil( %DB100.DBX2.7 )
   END_RUNG
   RUNG wire#w2
      R_Coil( %DB100.DBX4.7 )
   END_RUNG
   RUNG wire#w2
      R_Coil( %DB100.DBX6.7 )
   END_RUNG
   // the same network as SCL:
   IF "AlwaysTRUE" AND NOT "IsRem" THEN "dbzarządzanie".sterowanie_1.tryb_automat := FALSE; END_IF;
   #_w1 := "AlwaysTRUE" AND NOT "dbzarządzanie".sterowanie_1.tryb_automat;
   #_w2 := #_w1 AND NOT "Memeory_ResAut";   // rising edge
   "Memeory_ResAut" := #_w1;
   IF #_w2 THEN
       %DB100.DBX0.7 := FALSE;
       %DB100.DBX2.7 := FALSE;
       %DB100.DBX4.7 := FALSE;
       %DB100.DBX6.7 := FALSE;
   END_IF;
END_REGION

REGION Network 10
   RUNG wire#powerrail
      Contact( "AlwaysTRUE" )
      I_Contact( "IsRem" )
      wire#w1
      R_Coil( %DB100.DBX0.7 )
   END_RUNG
   RUNG wire#w1
      R_Coil( %DB100.DBX2.7 )
   END_RUNG
   RUNG wire#w1
      R_Coil( %DB100.DBX4.7 )
   END_RUNG
   RUNG wire#w1
      R_Coil( %DB100.DBX6.7 )
   END_RUNG
   // the same network as SCL:
   IF "AlwaysTRUE" AND NOT "IsRem" THEN
       %DB100.DBX0.7 := FALSE;
       %DB100.DBX2.7 := FALSE;
       %DB100.DBX4.7 := FALSE;
       %DB100.DBX6.7 := FALSE;
   END_IF;
END_REGION

REGION Network 11: PID is auto = 3 , mamual =4
   // PID tryb manualnye = ON/OFF
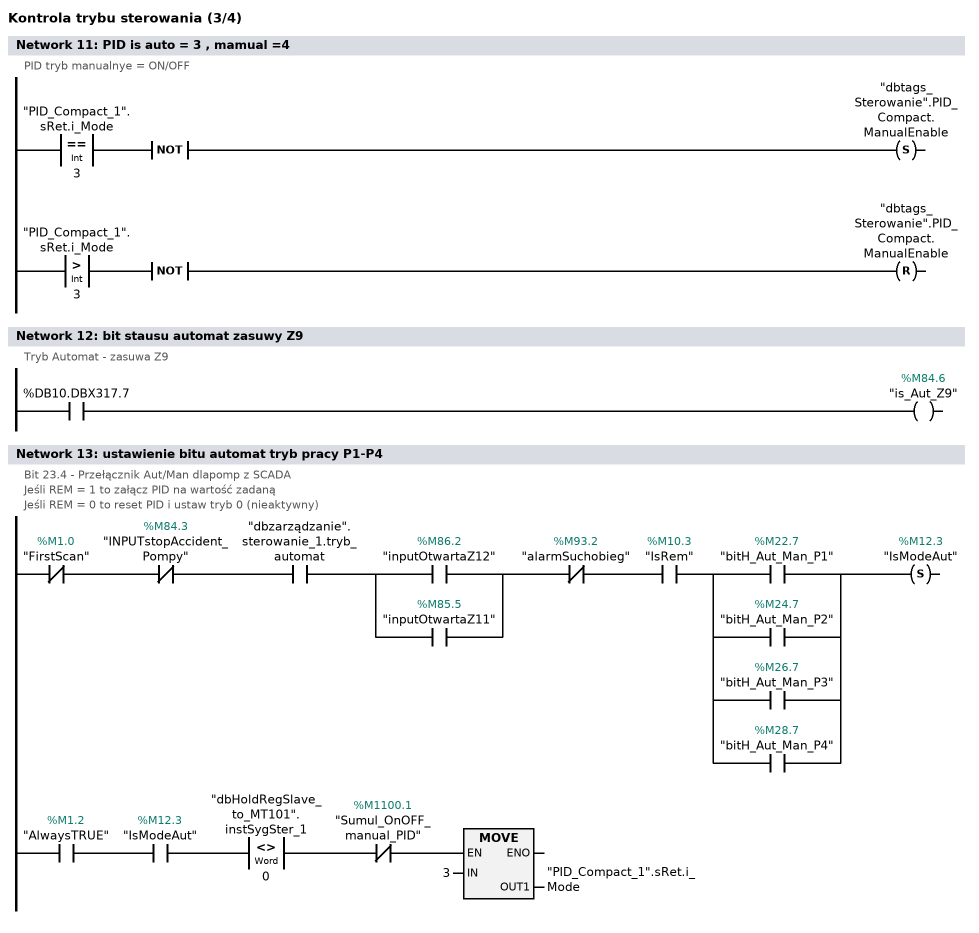
   RUNG wire#powerrail
      { S7_Templates := "SrcType := Int" } EQ_Contact(in1 := "PID_Compact_1".sRet.i_Mode, in2 := 3)
      Not()
      S_Coil( "dbtags_Sterowanie".PID_Compact.ManualEnable )
   END_RUNG
   RUNG wire#powerrail
      { S7_Templates := "SrcType := Int" } GT_Contact(in1 := "PID_Compact_1".sRet.i_Mode, in2 := 3)
      Not()
      R_Coil( "dbtags_Sterowanie".PID_Compact.ManualEnable )
   END_RUNG
   // the same network as SCL:
   IF NOT ("PID_Compact_1".sRet.i_Mode = 3) THEN
       "dbtags_Sterowanie".PID_Compact.ManualEnable := TRUE;
   END_IF;
   IF NOT ("PID_Compact_1".sRet.i_Mode > 3) THEN
       "dbtags_Sterowanie".PID_Compact.ManualEnable := FALSE;
   END_IF;
END_REGION

REGION Network 12: bit stausu automat zasuwy Z9
   // Tryb Automat - zasuwa Z9
   RUNG wire#powerrail
      Contact( %DB10.DBX317.7 )
      Coil( "is_Aut_Z9" )
   END_RUNG
   // the same network as SCL:
   "is_Aut_Z9" := %DB10.DBX317.7;
END_REGION

REGION Network 13: ustawienie bitu automat tryb pracy P1-P4
   // Bit 23.4 - Przełącznik Aut/Man dlapomp z SCADA
   // Jeśli REM = 1 to załącz PID na wartość zadaną
   // Jeśli REM = 0 to reset PID i ustaw tryb 0 (nieaktywny)
   RUNG wire#powerrail
      I_Contact( "FirstScan" )
      I_Contact( "INPUTstopAccident_Pompy" )
      Contact( "dbzarządzanie".sterowanie_1.tryb_automat )
      wire#w1
      Contact( "inputOtwartaZ12" )
      wire#w2
      I_Contact( "alarmSuchobieg" )
      Contact( "IsRem" )
      wire#w3
      Contact( "bitH_Aut_Man_P1" )
      wire#w4
      S_Coil( "IsModeAut" )
   END_RUNG
   RUNG wire#w1
      Contact( "inputOtwartaZ11" )
   END_RUNG wire#w2
   RUNG wire#w3
      Contact( "bitH_Aut_Man_P2" )
   END_RUNG wire#w4
   RUNG wire#w3
      Contact( "bitH_Aut_Man_P3" )
   END_RUNG wire#w4
   RUNG wire#w3
      Contact( "bitH_Aut_Man_P4" )
   END_RUNG wire#w4
   RUNG wire#powerrail
      Contact( "AlwaysTRUE" )
      Contact( "IsModeAut" )
      { S7_Templates := "SrcType := Word" } NE_Contact(in1 := "dbHoldRegSlave_to_MT101".instSygSter_1, in2 := 0)
      I_Contact( "Sumul_OnOFF_manual_PID" )
      { S7_GenerateENO := "TRUE" } Move(in := 3, out1 => "PID_Compact_1".sRet.i_Mode)
   END_RUNG
   // the same network as SCL:
   IF NOT "FirstScan" AND NOT "INPUTstopAccident_Pompy" AND "dbzarządzanie".sterowanie_1.tryb_automat AND ("inputOtwartaZ12" OR "inputOtwartaZ11") AND NOT "alarmSuchobieg" AND "IsRem" AND ("bitH_Aut_Man_P1" OR "bitH_Aut_Man_P2" OR "bitH_Aut_Man_P3" OR "bitH_Aut_Man_P4") THEN
       "IsModeAut" := TRUE;
   END_IF;
   IF "AlwaysTRUE" AND "IsModeAut" AND ("dbHoldRegSlave_to_MT101".instSygSter_1 <> 0) AND NOT "Sumul_OnOFF_manual_PID" THEN
       "PID_Compact_1".sRet.i_Mode := 3;
   END_IF;
END_REGION

REGION Network 14: Reset bitu tryb pracy automat pomp
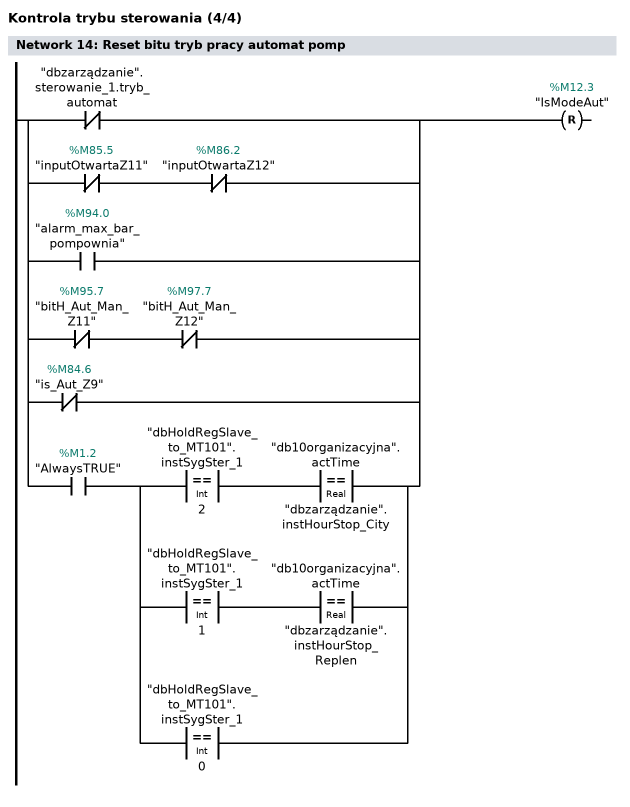
   RUNG wire#powerrail
      I_Contact( "dbzarządzanie".sterowanie_1.tryb_automat )
      wire#w1
      R_Coil( "IsModeAut" )
   END_RUNG
   RUNG wire#powerrail
      I_Contact( "inputOtwartaZ11" )
      I_Contact( "inputOtwartaZ12" )
   END_RUNG wire#w1
   RUNG wire#powerrail
      Contact( "alarm_max_bar_pompownia" )
   END_RUNG wire#w1
   RUNG wire#powerrail
      I_Contact( "bitH_Aut_Man_Z11" )
      I_Contact( "bitH_Aut_Man_Z12" )
   END_RUNG wire#w1
   RUNG wire#powerrail
      I_Contact( "is_Aut_Z9" )
   END_RUNG wire#w1
   RUNG wire#powerrail
      Contact( "AlwaysTRUE" )
      wire#w2
      { S7_Templates := "SrcType := Int" } EQ_Contact(in1 := "dbHoldRegSlave_to_MT101".instSygSter_1, in2 := 2)
      { S7_Templates := "SrcType := Real" } EQ_Contact(in1 := "db10organizacyjna".actTime, in2 := "dbzarządzanie".instHourStop_City)
   END_RUNG wire#w1
   RUNG wire#w2
      { S7_Templates := "SrcType := Int" } EQ_Contact(in1 := "dbHoldRegSlave_to_MT101".instSygSter_1, in2 := 1)
      { S7_Templates := "SrcType := Real" } EQ_Contact(in1 := "db10organizacyjna".actTime, in2 := "dbzarządzanie".instHourStop_Replen)
   END_RUNG wire#w1
   RUNG wire#w2
      { S7_Templates := "SrcType := Int" } EQ_Contact(in1 := "dbHoldRegSlave_to_MT101".instSygSter_1, in2 := 0)
   END_RUNG wire#w1
   // the same network as SCL:
   IF NOT "dbzarządzanie".sterowanie_1.tryb_automat OR (NOT "inputOtwartaZ11" AND NOT "inputOtwartaZ12") OR "alarm_max_bar_pompownia" OR (NOT "bitH_Aut_Man_Z11" AND NOT "bitH_Aut_Man_Z12") OR NOT "is_Aut_Z9" OR ("AlwaysTRUE" AND ((("dbHoldRegSlave_to_MT101".instSygSter_1 = 2) AND ("db10organizacyjna".actTime = "dbzarządzanie".instHourStop_City)) OR (("dbHoldRegSlave_to_MT101".instSygSter_1 = 1) AND ("db10organizacyjna".actTime = "dbzarządzanie".instHourStop_Replen)) OR ("dbHoldRegSlave_to_MT101".instSygSter_1 = 0))) THEN
       "IsModeAut" := FALSE;
   END_IF;
END_REGION
END_FUNCTION

FUNCTION_BLOCK "Kontrola przyrostu ciśnieniea"   // FB3, LAD
TITLE = Kalkulacja przyrostu ciśnienia w czasie
{ S7_Optimized_Access := 'TRUE' }
AUTHOR : RTecmer
FAMILY : PID
VERSION : 0.1
// Funkcja ustala czy następuje przyrost ciśnienia, spadek, równowaga. Pomiar dokonywany jest w ustalonym czasie. W zależności od wyliceń ustawiany jest znacznik, który w funkcji Switch_Motor_Extra dopuszcza lub blokuje uruchomienie dodatkowej pompy
// stored: AutoNumber true, IsIECCheckEnabled false, IsRetainMemResEnabled false, MemoryReserve 500, SetENOAutomatically false, UDAEnableTagReadback false
   VAR_INPUT
      "50Hz" : Bool;   // Znacznik 50Hz
      "Set_O2-PID" : Real;   // Zadana wartość ciśnienia [bar]
      Current_bar_1 : Real;   // aktualne ciśnienie
   END_VAR
   VAR_OUTPUT
      Increase_in_value : Bool;   // Wzwrost wartości bar w jednostce czasu
   END_VAR
   VAR_IN_OUT
      Edge1_Hz : Bool;   // Pamięć zbocza dla pierwszego odczytu
      Edge2_Hz : Bool;   // Pamięć zbocza dla drugiego odczytu
      Data_sek_1 : Int;   // Licznik sekund dla pierwszego odczytu
      Data_sek_2 : Int;   // Licznik sekund dla drugiego odczytu
      Pause_1 : Bool;   // Wstrzymanie dla pierwszego czasu
      Pause_2 : Bool;   // wstrzymanie dla drugiego czasu
   END_VAR
   VAR_TEMP   // added for the SCL form of the ladder/FBD networks
      _w1 : Bool;
      _w2 : Bool;
   END_VAR
BEGIN

REGION Network 1: Wstrzymanie dla pierwszego czasu
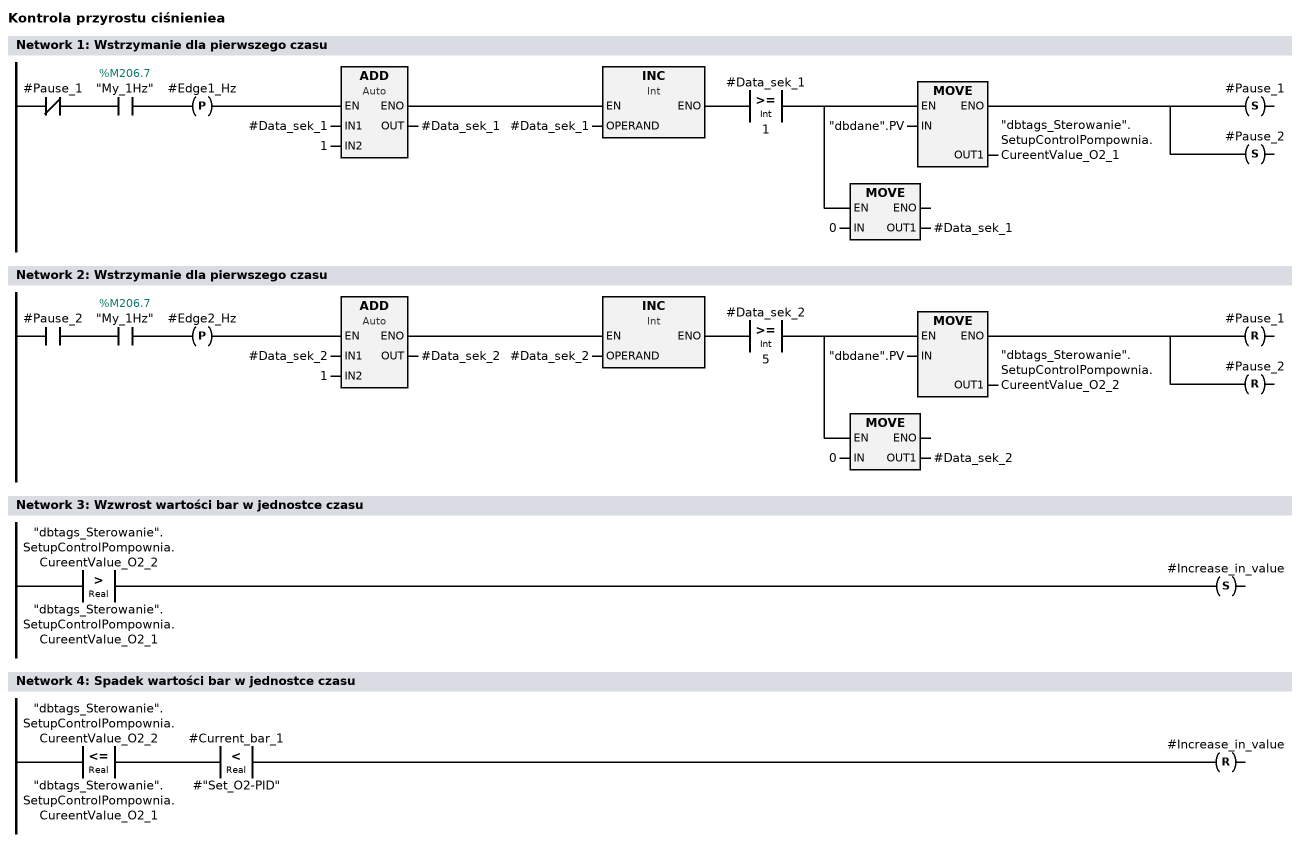
   RUNG wire#powerrail
      I_Contact( #Pause_1 )
      Contact( "My_1Hz" )
      P_Trig( #Edge1_Hz )
      { S7_GenerateENO := "TRUE" } Add(in1 := #Data_sek_1, in2 := 1, out => #Data_sek_1)
      { S7_Templates := "DestType := Int"; S7_GenerateENO := "TRUE" } Inc( #Data_sek_1 )
      { S7_Templates := "SrcType := Int" } GE_Contact(in1 := #Data_sek_1, in2 := 1)
      wire#w1
      { S7_GenerateENO := "TRUE" } Move(in := "dbdane".PV, out1 => "dbtags_Sterowanie".SetupControlPompownia.CureentValue_O2_1)
      wire#w2
      S_Coil( #Pause_1 )
   END_RUNG
   RUNG wire#w2
      S_Coil( #Pause_2 )
   END_RUNG
   RUNG wire#w1
      { S7_GenerateENO := "TRUE" } Move(in := 0, out1 => #Data_sek_1)
   END_RUNG
   // the same network as SCL:
   // ENO of a box is taken as its EN; it also drops when the box reports an error
   #_w1 := NOT #Pause_1 AND "My_1Hz";
   #_w2 := #_w1 AND NOT #Edge1_Hz;   // rising edge
   #Edge1_Hz := #_w1;
   IF #_w2 THEN
       #Data_sek_1 := #Data_sek_1 + 1;
       #Data_sek_1 := #Data_sek_1 + 1;
   END_IF;
   IF #_w2 AND (#Data_sek_1 >= 1) THEN
       "dbtags_Sterowanie".SetupControlPompownia.CureentValue_O2_1 := "dbdane".PV;
       #Pause_1 := TRUE;
       #Pause_2 := TRUE;
       #Data_sek_1 := 0;
   END_IF;
END_REGION

REGION Network 2: Wstrzymanie dla pierwszego czasu
   RUNG wire#powerrail
      Contact( #Pause_2 )
      Contact( "My_1Hz" )
      P_Trig( #Edge2_Hz )
      { S7_GenerateENO := "TRUE" } Add(in1 := #Data_sek_2, in2 := 1, out => #Data_sek_2)
      { S7_Templates := "DestType := Int"; S7_GenerateENO := "TRUE" } Inc( #Data_sek_2 )
      { S7_Templates := "SrcType := Int" } GE_Contact(in1 := #Data_sek_2, in2 := 5)
      wire#w1
      { S7_GenerateENO := "TRUE" } Move(in := "dbdane".PV, out1 => "dbtags_Sterowanie".SetupControlPompownia.CureentValue_O2_2)
      wire#w2
      R_Coil( #Pause_1 )
   END_RUNG
   RUNG wire#w2
      R_Coil( #Pause_2 )
   END_RUNG
   RUNG wire#w1
      { S7_GenerateENO := "TRUE" } Move(in := 0, out1 => #Data_sek_2)
   END_RUNG
   // the same network as SCL:
   // ENO of a box is taken as its EN; it also drops when the box reports an error
   #_w1 := #Pause_2 AND "My_1Hz";
   #_w2 := #_w1 AND NOT #Edge2_Hz;   // rising edge
   #Edge2_Hz := #_w1;
   IF #_w2 THEN
       #Data_sek_2 := #Data_sek_2 + 1;
       #Data_sek_2 := #Data_sek_2 + 1;
   END_IF;
   IF #_w2 AND (#Data_sek_2 >= 5) THEN
       "dbtags_Sterowanie".SetupControlPompownia.CureentValue_O2_2 := "dbdane".PV;
       #Pause_1 := FALSE;
       #Pause_2 := FALSE;
       #Data_sek_2 := 0;
   END_IF;
END_REGION

REGION Network 3: Wzwrost wartości bar w jednostce czasu
   RUNG wire#powerrail
      { S7_Templates := "SrcType := Real" } GT_Contact(in1 := "dbtags_Sterowanie".SetupControlPompownia.CureentValue_O2_2, in2 := "dbtags_Sterowanie".SetupControlPompownia.CureentValue_O2_1)
      S_Coil( #Increase_in_value )
   END_RUNG
   // the same network as SCL:
   IF "dbtags_Sterowanie".SetupControlPompownia.CureentValue_O2_2 > "dbtags_Sterowanie".SetupControlPompownia.CureentValue_O2_1 THEN
       #Increase_in_value := TRUE;
   END_IF;
END_REGION

REGION Network 4: Spadek wartości bar w jednostce czasu
   RUNG wire#powerrail
      { S7_Templates := "SrcType := Real" } LE_Contact(in1 := "dbtags_Sterowanie".SetupControlPompownia.CureentValue_O2_2, in2 := "dbtags_Sterowanie".SetupControlPompownia.CureentValue_O2_1)
      { S7_Templates := "SrcType := Real" } LT_Contact(in1 := #Current_bar_1, in2 := #"Set_O2-PID")
      R_Coil( #Increase_in_value )
   END_RUNG
   // the same network as SCL:
   IF ("dbtags_Sterowanie".SetupControlPompownia.CureentValue_O2_2 <= "dbtags_Sterowanie".SetupControlPompownia.CureentValue_O2_1) AND (#Current_bar_1 < #"Set_O2-PID") THEN
       #Increase_in_value := FALSE;
   END_IF;
END_REGION
END_FUNCTION_BLOCK

FUNCTION_BLOCK "Byte status pomp"
TITLE = Calculation Byte Status Pomp
{ S7_Optimized_Access := 'TRUE' }
AUTHOR : rtecmer
VERSION : 0.1
//Byte określający ile napędów dostępnych. Wykorzystywany do blokowania przełączenia na sieć ostatniej dostępnej dmuchawy.

BEGIN
	(*
	//=============================================================================
	//(JZWiK S.A Radosław Tecmer)
	//(c)Copyright (2021) All Rights Reserved
	//-----------------------------------------------------------------------------
	//Testowane z:   (system docelowy z  FW 4.4)
	//Pakiet inżynierski:   TIA Portal (V14 Sp1 Update 9)
	//Ograniczenia:  ( - )
	//Wymagania:  (minimalne S7-1200 CPU 1215C FW 4.2 .)
	//Funkcjonalnośc: (Byte statusu napędów P1-P4 Pompowna )
	//-----------------------------------------------------------------------------
	//Zmainy wprowadzone:
	//Wersja  Data       Osoba wprowadzająca zmiany - ekspert
	//01.00.00 17.11.2021 (Tecmer Radosław - twórca) Pieresza wersja 01.00.00
	//=============================================================================
	*)
	
	REGION przekazanie satusu P1 P2 P3 P4 Z11 Z12  do znacznika
	  //przekazanie
	  // P1 Przekazanie Byte H ststusu do Byte znacznika 
	  "ByteH_Status_P1" := %DB100.DBB1;
	  // P2 Przekazanie Byte H ststusu do Byte znacznika 
	  "ByteH_Status_P2" := %DB100.DBB3;
	  // P3 Przekazanie Byte H ststusu do Byte znacznika 
	  "ByteH_Status_P3" := %DB100.DBB5;
	  // P4 Przekazanie Byte H ststusu do Byte znacznika 
	  "ByteH_Status_P4" := %DB100.DBB7;
	  
	  
	END_REGION
	
	IF "IsReady_P1" AND "bitH_Aut_Man_P1" AND (NOT "IsRunNetwork_P1")AND (NOT "IsRunInverter_P1") THEN
	  // Przekaż wartość 1 gdy gotowość P1
	  "dbzarządzanie".sterowanie_1.aktywna_P1:= TRUE;
	ELSE
	  "dbzarządzanie".sterowanie_1.aktywna_P1 := FALSE;
	END_IF;
	
	"activePump_P1" :="dbzarządzanie".sterowanie_1.aktywna_P1 ;
	
	
	IF "IsReady_P2" AND "bitH_Aut_Man_P2" AND (NOT "IsRunNetwork_P2")AND (NOT "IsRunInverter_P2") THEN
	  // Przekaż wartość 1 gdy gotowość P2
	  "dbzarządzanie".sterowanie_1.aktywna_P2 := TRUE;
	ELSE
	  "dbzarządzanie".sterowanie_1.aktywna_P2 := FALSE;
	END_IF;
	
	"activePump_P2" :="dbzarządzanie".sterowanie_1.aktywna_P2;
	
	IF "IsReady_P3" AND "bitH_Aut_Man_P3" AND (NOT "IsRunNetwork_P3")AND (NOT "IsRunInverter_P3") THEN
	  // Przekaż wartość 1 gdy gotowość P3
	  "dbzarządzanie".sterowanie_1.aktywna_P3 := TRUE;
	ELSE
	  "dbzarządzanie".sterowanie_1.aktywna_P3 := FALSE;
	END_IF;
	
	"activePump_P3" :="dbzarządzanie".sterowanie_1.aktywna_P3 ;
	
	IF "IsReady_P4" AND "bitH_Aut_Man_P4" AND (NOT "IsRunNetwork_P4")AND (NOT "IsRunInverter_P4") THEN
	  // Przekaż wartość 1 gdy gotowość P4
	  "dbzarządzanie".sterowanie_1.aktywna_P4  := TRUE;
	ELSE
	  "dbzarządzanie".sterowanie_1.aktywna_P4  := FALSE;
	END_IF;
	
	"activePump_P4" :="dbzarządzanie".sterowanie_1.aktywna_P4 ;
	
	
	
END_FUNCTION_BLOCK

FUNCTION "Opóżnienie wiodącej_dodatkowych" : Void   // FC26, LAD
TITLE = Przełącznik czasu do startu dodatkowej
{ S7_Optimized_Access := 'TRUE' }
AUTHOR : rtecmer
VERSION : 0.1
// Przełączanie wartości czasu startu napędu dodatkowego w zależności od przepływu
// stored: AutoNumber true, IsIECCheckEnabled false, SetENOAutomatically false, UDAEnableTagReadback false
BEGIN

REGION Network 1
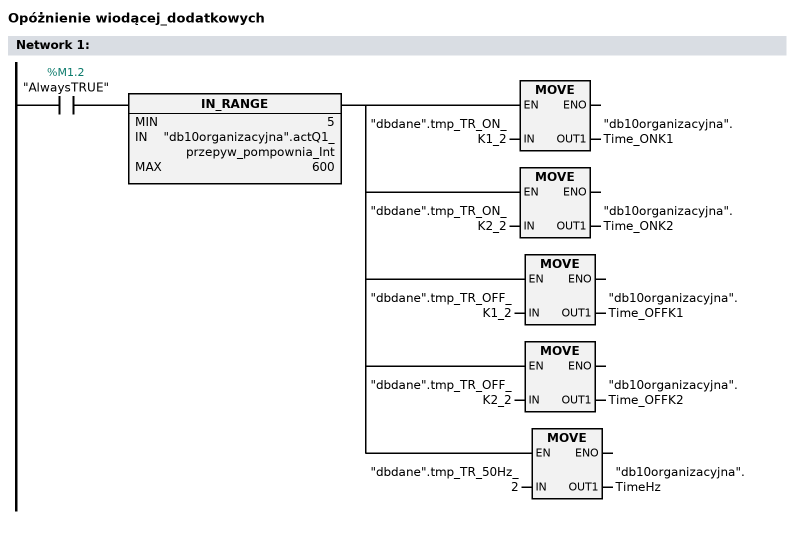
   RUNG wire#powerrail
      Contact( "AlwaysTRUE" )
      { S7_Templates := "SrcType := Int" } InRange(min := 5, in := "db10organizacyjna".actQ1_przepyw_pompownia_Int, max := 600)
      wire#w1
      Move(in := "dbdane".tmp_TR_ON_K1_2, out1 => "db10organizacyjna".Time_ONK1)
   END_RUNG
   RUNG wire#w1
      Move(in := "dbdane".tmp_TR_ON_K2_2, out1 => "db10organizacyjna".Time_ONK2)
   END_RUNG
   RUNG wire#w1
      Move(in := "dbdane".tmp_TR_OFF_K1_2, out1 => "db10organizacyjna".Time_OFFK1)
   END_RUNG
   RUNG wire#w1
      Move(in := "dbdane".tmp_TR_OFF_K2_2, out1 => "db10organizacyjna".Time_OFFK2)
   END_RUNG
   RUNG wire#w1
      Move(in := "dbdane".tmp_TR_50Hz_2, out1 => "db10organizacyjna".TimeHz)
   END_RUNG
   // the same network as SCL:
   IF "AlwaysTRUE" AND (5 <= "db10organizacyjna".actQ1_przepyw_pompownia_Int) AND ("db10organizacyjna".actQ1_przepyw_pompownia_Int <= 600) THEN
       "db10organizacyjna".Time_ONK1 := "dbdane".tmp_TR_ON_K1_2;
       "db10organizacyjna".Time_ONK2 := "dbdane".tmp_TR_ON_K2_2;
       "db10organizacyjna".Time_OFFK1 := "dbdane".tmp_TR_OFF_K1_2;
       "db10organizacyjna".Time_OFFK2 := "dbdane".tmp_TR_OFF_K2_2;
       "db10organizacyjna".TimeHz := "dbdane".tmp_TR_50Hz_2;
   END_IF;
END_REGION
END_FUNCTION

FUNCTION_BLOCK "Sterowanie pompami dodatkowymi"   // FB1, LAD
TITLE = Funkcja ustawiająca załączenie regulatora i ilość pomp dodatkowych
{ S7_Optimized_Access := 'TRUE' }
AUTHOR : RTecmer
FAMILY : Ster
VERSION : 0.1
// Sterowanie pompami
// stored: AutoNumber true, IsIECCheckEnabled false, IsRetainMemResEnabled false, MemoryReserve 500, SetENOAutomatically false, UDAEnableTagReadback false
   VAR_INPUT
      daneMV { ExternalAccessible := 'False'; ExternalVisible := 'False'; ExternalWritable := 'False'} : Real;   // Aktualne Hz na wyjściu QW64 - zadane Hz
      trybPracyPID { ExternalAccessible := 'False'; ExternalVisible := 'False'; ExternalWritable := 'False'} : Int;   // Aktualny tryb pracy regulatora PID1 [0-wyłącznony, 1- Pretuning, 2- Manual fine tuning, 3- praca auto, 4- Manual mode
      IsMode_Aut { ExternalAccessible := 'False'; ExternalVisible := 'False'; ExternalWritable := 'False'} : Bool;   // Tryb pracy układu sterowania
      IsReady_F1 { ExternalAccessible := 'False'; ExternalVisible := 'False'; ExternalWritable := 'False'} : Bool;
      InputWarning_H_PID { ExternalAccessible := 'False'; ExternalVisible := 'False'; ExternalWritable := 'False'} : Bool;   // Oszczerzenie górny limit
      InputWarning_L_PID { ExternalAccessible := 'False'; ExternalVisible := 'False'; ExternalWritable := 'False'} : Bool;   // Oczszczerzenie dolny limit
      Timer_K1 { ExternalAccessible := 'False'; ExternalVisible := 'False'; ExternalWritable := 'False'} : Time;   // Opóźnienie do załączenie K1
      Timer_K2 { ExternalAccessible := 'False'; ExternalVisible := 'False'; ExternalWritable := 'False'} : Time;   // Opóźnienie do załaczenia K2
      Timer_K3 : Time;   // Opóźnienie do załaczenia K3
      Timer_OFF_K1 { ExternalAccessible := 'False'; ExternalVisible := 'False'; ExternalWritable := 'False'} : Time;
      Timer_OFF_K2 { ExternalAccessible := 'False'; ExternalVisible := 'False'; ExternalWritable := 'False'} : Time;
      Timer_OFF_K3 { ExternalAccessible := 'False'; ExternalVisible := 'False'; ExternalWritable := 'False'} : Time;
      Time_50Hz { ExternalAccessible := 'False'; ExternalVisible := 'False'; ExternalWritable := 'False'} : Time;   // Histereza na ustawienie flagi Hz50
      IsAuto_P1 : Bool;   // Sygnał sterowanie automatyczne
      IsAuto_P2 : Bool;   // Sygnał sterowanie automatyczne
      IsAuto_P3 : Bool;   // Sygnał sterowanie automatyczne
      IsAuto_P4 : Bool;   // Sygnał sterowanie automatyczne
      Mem_K1 : Bool;   // Flaga pamięci załączenia K1 od WarningLowLimit
      IsIncrease : Bool;   // Flaga przyrostu ciśnienia w jednostce czasu
      CureentQ1 : Word;   // Przepływ pompownia
      IsRunInverterMA : Bool;   // Potwierdzenie falownika MA
      IsRunInverterMB : Bool := false;   // Potwierdzenie falownika MA
      IsRunInverterMC : Bool := false;   // Potwierdzenie falownika MA
      IsRunInverterMD : Bool := false;   // Potwierdzenie falownika MA
      IsReady_MA : Bool;   // Potwierdzenie gotowości pompa 1 dodatkowa
      IsReady_MB : Bool := false;   // Potwierdzenie gotowości pompa 2 dodatkowa
      IsReady_MC : Bool := false;   // Potwierdzenie gotowości pompa wiodąca
      IsReady_MD : Bool := false;   // Potwierdzenie gotowości pompa 3 dodatkowa
      Rst_Motor2_Alarm : Bool;   // Znacznik wyłaczenia od alarmu dodatkowej 1
      Rst_Motor3_Alarm : Bool;   // Znacznik wyłączenia od alarmu dodatkowej 2
      Rst_Motor4_Alarm : Bool;   // Znacznik wyłączenia od alarmu dodatkowej 3
      correction_reset_K1 : Real;   // Wspólczynnik pomniejszenia wyliczanego cisnienie napotrzeby wyłączenia dodatowej
      correction_reset_K2 : Real;   // Wspólczynnik pomniejszenia wyliczanego ciśnienia napotrzeby wyłączenia dodatowej
   END_VAR
   VAR_IN_OUT
      Set_K1 { ExternalWritable := 'False'} : Bool;   // Dostaw 1 pompę dodatkową
      Set_K2 { ExternalWritable := 'False'} : Bool;   // Dostaw 2 dodatkową
      Set_K3 : Bool;   // Dostaw 3 dodatkową
      Set_K4 { ExternalWritable := 'False'} : Bool;   // Uruchom Regulator PID
   END_VAR
   VAR
      Temp_bar_OFF { ExternalAccessible := 'False'; ExternalVisible := 'False'; ExternalWritable := 'False'} : Real;   // Wartosc cisnienia do wyłączenia szybkiego
      reset_Value_K1 { ExternalAccessible := 'False'; ExternalVisible := 'False'; ExternalWritable := 'False'} : Real;   // Wartość bar do wyłączenie dodatkowej nr 1
      reset_Value_K2 { ExternalAccessible := 'False'; ExternalVisible := 'False'; ExternalWritable := 'False'} : Real;   // Wartość bar do wyłączenie dodatkowej nr 2
      reset_value_K3 { ExternalAccessible := 'False'; ExternalVisible := 'False'; ExternalWritable := 'False'} : Real;   // Wartość bar do wyłączenie dodatkowej nr 3
      table_index { ExternalAccessible := 'False'; ExternalVisible := 'False'; ExternalWritable := 'False'} : Int;   // Index tablicy z stałymi parametrami Hz
      WarningHigbar { ExternalAccessible := 'False'; ExternalVisible := 'False'; ExternalWritable := 'False'} : Real;   // Wartośc stała napotrzeby wyłączenia dodatkowej
      notManau { ExternalAccessible := 'False'; ExternalVisible := 'False'; ExternalWritable := 'False'} : Bool;   // Przynajmniej jedna w trybie "Autmat"
      temp_reset_value_K3 { ExternalAccessible := 'False'; ExternalVisible := 'False'; ExternalWritable := 'False'} : Real;
      is_correctio_bar { ExternalAccessible := 'False'; ExternalVisible := 'False'; ExternalWritable := 'False'} : Bool;   // znacznik wzrostu ciśnienia
   END_VAR
   VAR_TEMP   // added for the SCL form of the ladder/FBD networks
      _w1 : Bool;
      _w2 : Bool;
   END_VAR
BEGIN

REGION Network 1: Histereza na ustawienie flagi 50_Hz
   // Odmierzanie zwłoki na ustawienie znacznika "50Hz"
   // znacznik "notManau" - blokuje ustawienie znacznika FC2_Set_50Hz gdy brak wolnej pompy dodatkowej.
   // eleiminuje przełączenie się ostatniej pompy na SIEĆ
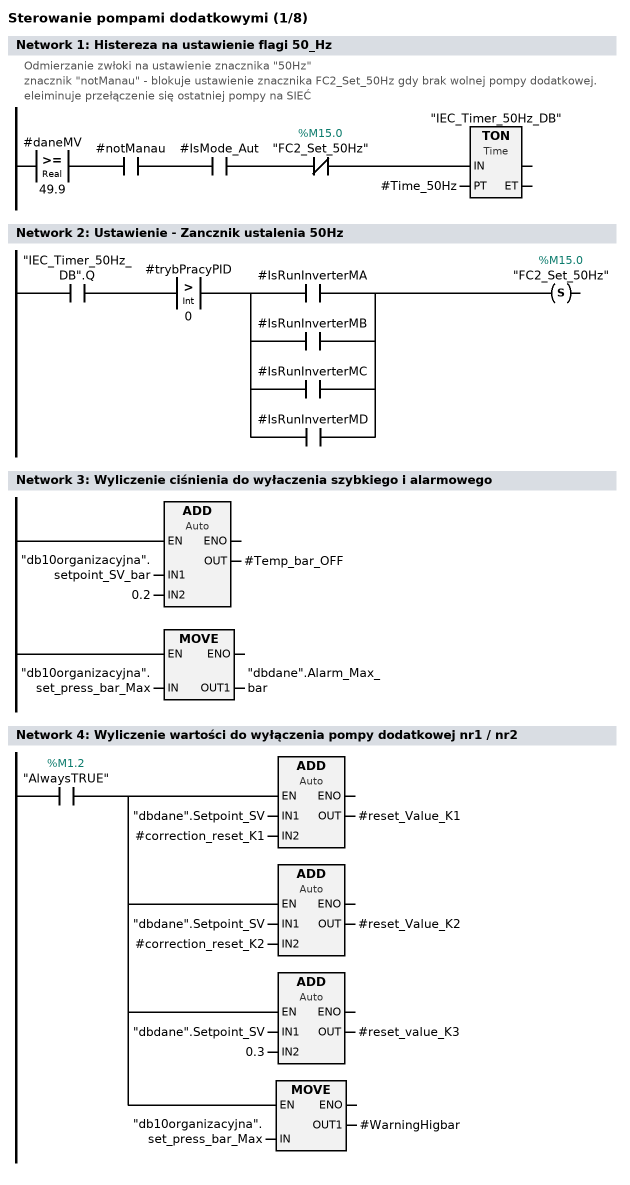
   RUNG wire#powerrail
      { S7_Templates := "SrcType := Real" } GE_Contact(in1 := #daneMV, in2 := 49.9)
      Contact( #notManau )
      Contact( #IsMode_Aut )
      I_Contact( "FC2_Set_50Hz" )
      { S7_Templates := "time_type := Time" } "IEC_Timer_50Hz_DB".TON(pt := #Time_50Hz, et =>)
   END_RUNG
   // the same network as SCL:
   "IEC_Timer_50Hz_DB".TON(IN := (#daneMV >= 49.9) AND #notManau AND #IsMode_Aut AND NOT "FC2_Set_50Hz",
                           PT := #Time_50Hz);
END_REGION

REGION Network 2: Ustawienie - Zancznik ustalenia 50Hz
   RUNG wire#powerrail
      Contact( "IEC_Timer_50Hz_DB".Q )
      { S7_Templates := "SrcType := Int" } GT_Contact(in1 := #trybPracyPID, in2 := 0)
      wire#w1
      Contact( #IsRunInverterMA )
      wire#w2
      S_Coil( "FC2_Set_50Hz" )
   END_RUNG
   RUNG wire#w1
      Contact( #IsRunInverterMB )
   END_RUNG wire#w2
   RUNG wire#w1
      Contact( #IsRunInverterMC )
   END_RUNG wire#w2
   RUNG wire#w1
      Contact( #IsRunInverterMD )
   END_RUNG wire#w2
   // the same network as SCL:
   IF "IEC_Timer_50Hz_DB".Q AND (#trybPracyPID > 0) AND (#IsRunInverterMA OR #IsRunInverterMB OR #IsRunInverterMC OR #IsRunInverterMD) THEN
       "FC2_Set_50Hz" := TRUE;
   END_IF;
END_REGION

REGION Network 3: Wyliczenie ciśnienia do wyłaczenia szybkiego i alarmowego
   RUNG wire#powerrail
      { S7_GenerateENO := "TRUE" } Add(in1 := "db10organizacyjna".setpoint_SV_bar, in2 := 0.2, out => #Temp_bar_OFF)
   END_RUNG
   RUNG wire#powerrail
      Move(in := "db10organizacyjna".set_press_bar_Max, out1 => "dbdane".Alarm_Max_bar)
   END_RUNG
   // the same network as SCL:
   #Temp_bar_OFF := "db10organizacyjna".setpoint_SV_bar + 0.2;
   "dbdane".Alarm_Max_bar := "db10organizacyjna".set_press_bar_Max;
END_REGION

REGION Network 4: Wyliczenie wartości do wyłączenia pompy dodatkowej nr1 / nr2
   RUNG wire#powerrail
      Contact( "AlwaysTRUE" )
      wire#w1
      Add(in1 := "dbdane".Setpoint_SV, in2 := #correction_reset_K1, out => #reset_Value_K1)
   END_RUNG
   RUNG wire#w1
      Add(in1 := "dbdane".Setpoint_SV, in2 := #correction_reset_K2, out => #reset_Value_K2)
   END_RUNG
   RUNG wire#w1
      Add(in1 := "dbdane".Setpoint_SV, in2 := 0.3, out => #reset_value_K3)
   END_RUNG
   RUNG wire#w1
      Move(in := "db10organizacyjna".set_press_bar_Max, out1 => #WarningHigbar)
   END_RUNG
   // the same network as SCL:
   IF "AlwaysTRUE" THEN
       #reset_Value_K1 := "dbdane".Setpoint_SV + #correction_reset_K1;
       #reset_Value_K2 := "dbdane".Setpoint_SV + #correction_reset_K2;
       #reset_value_K3 := "dbdane".Setpoint_SV + 0.3;
       #WarningHigbar := "db10organizacyjna".set_press_bar_Max;
   END_IF;
END_REGION

REGION Network 5: Sprawdzenie dostepnej pompy
   // Jesli przynajmniej jedna dodatkwa dostepna w innym przypadku nie nastąpi dostawianie pomp dodatkowych
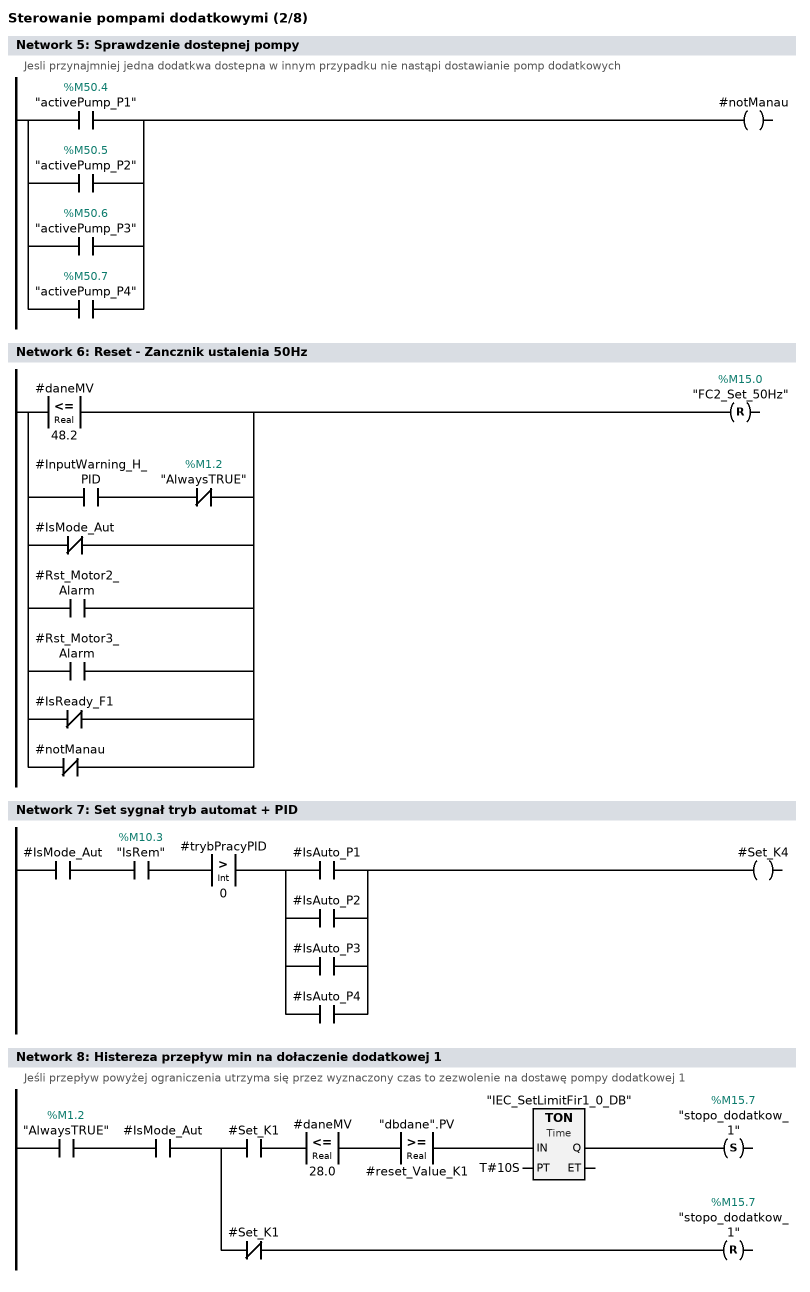
   RUNG wire#powerrail
      Contact( "activePump_P1" )
      wire#w1
      Coil( #notManau )
   END_RUNG
   RUNG wire#powerrail
      Contact( "activePump_P2" )
   END_RUNG wire#w1
   RUNG wire#powerrail
      Contact( "activePump_P3" )
   END_RUNG wire#w1
   RUNG wire#powerrail
      Contact( "activePump_P4" )
   END_RUNG wire#w1
   // the same network as SCL:
   #notManau := "activePump_P1" OR "activePump_P2" OR "activePump_P3" OR "activePump_P4";
END_REGION

REGION Network 6: Reset - Zancznik ustalenia 50Hz
   RUNG wire#powerrail
      { S7_Templates := "SrcType := Real" } LE_Contact(in1 := #daneMV, in2 := 48.2)
      wire#w1
      R_Coil( "FC2_Set_50Hz" )
   END_RUNG
   RUNG wire#powerrail
      Contact( #InputWarning_H_PID )
      I_Contact( "AlwaysTRUE" )
   END_RUNG wire#w1
   RUNG wire#powerrail
      I_Contact( #IsMode_Aut )
   END_RUNG wire#w1
   RUNG wire#powerrail
      Contact( #Rst_Motor2_Alarm )
   END_RUNG wire#w1
   RUNG wire#powerrail
      Contact( #Rst_Motor3_Alarm )
   END_RUNG wire#w1
   RUNG wire#powerrail
      I_Contact( #IsReady_F1 )
   END_RUNG wire#w1
   RUNG wire#powerrail
      I_Contact( #notManau )
   END_RUNG wire#w1
   // the same network as SCL:
   IF (#daneMV <= 48.2) OR (#InputWarning_H_PID AND NOT "AlwaysTRUE") OR NOT #IsMode_Aut OR #Rst_Motor2_Alarm OR #Rst_Motor3_Alarm OR NOT #IsReady_F1 OR NOT #notManau THEN
       "FC2_Set_50Hz" := FALSE;
   END_IF;
END_REGION

REGION Network 7: Set sygnał tryb automat + PID
   RUNG wire#powerrail
      Contact( #IsMode_Aut )
      Contact( "IsRem" )
      { S7_Templates := "SrcType := Int" } GT_Contact(in1 := #trybPracyPID, in2 := 0)
      wire#w1
      Contact( #IsAuto_P1 )
      wire#w2
      Coil( #Set_K4 )
   END_RUNG
   RUNG wire#w1
      Contact( #IsAuto_P2 )
   END_RUNG wire#w2
   RUNG wire#w1
      Contact( #IsAuto_P3 )
   END_RUNG wire#w2
   RUNG wire#w1
      Contact( #IsAuto_P4 )
   END_RUNG wire#w2
   // the same network as SCL:
   #Set_K4 := #IsMode_Aut AND "IsRem" AND (#trybPracyPID > 0) AND (#IsAuto_P1 OR #IsAuto_P2 OR #IsAuto_P3 OR #IsAuto_P4);
END_REGION

REGION Network 8: Histereza przepływ min na dołaczenie dodatkowej 1
   // Jeśli przepływ powyżej ograniczenia utrzyma się przez wyznaczony czas to zezwolenie na dostawę pompy dodatkowej 1
   RUNG wire#powerrail
      Contact( "AlwaysTRUE" )
      Contact( #IsMode_Aut )
      wire#w1
      Contact( #Set_K1 )
      { S7_Templates := "SrcType := Real" } LE_Contact(in1 := #daneMV, in2 := 28.0)
      { S7_Templates := "SrcType := Real" } GE_Contact(in1 := "dbdane".PV, in2 := #reset_Value_K1)
      { S7_Templates := "time_type := Time" } "IEC_SetLimitFir1_0_DB".TON(pt := T#10S, et =>)
      S_Coil( "stopo_dodatkow_1" )
   END_RUNG
   RUNG wire#w1
      I_Contact( #Set_K1 )
      R_Coil( "stopo_dodatkow_1" )
   END_RUNG
   // the same network as SCL:
   #_w1 := "AlwaysTRUE" AND #IsMode_Aut;
   "IEC_SetLimitFir1_0_DB".TON(IN := #_w1 AND #Set_K1 AND (#daneMV <= 28.0) AND ("dbdane".PV >= #reset_Value_K1),
                           PT := T#10S);
   IF "IEC_SetLimitFir1_0_DB".Q THEN "stopo_dodatkow_1" := TRUE; END_IF;
   IF #_w1 AND NOT #Set_K1 THEN "stopo_dodatkow_1" := FALSE; END_IF;
END_REGION

REGION Network 9: Kontrola przyrostu ciśnienia
   // Kontrola czasu przyrostu ciśnienia. Jeśli  nie osiągnieta równowaga do zadanego czasu IEC_Timer_PID_SetK1_Full_DB = 1 minuta to ustaw Q Timera.
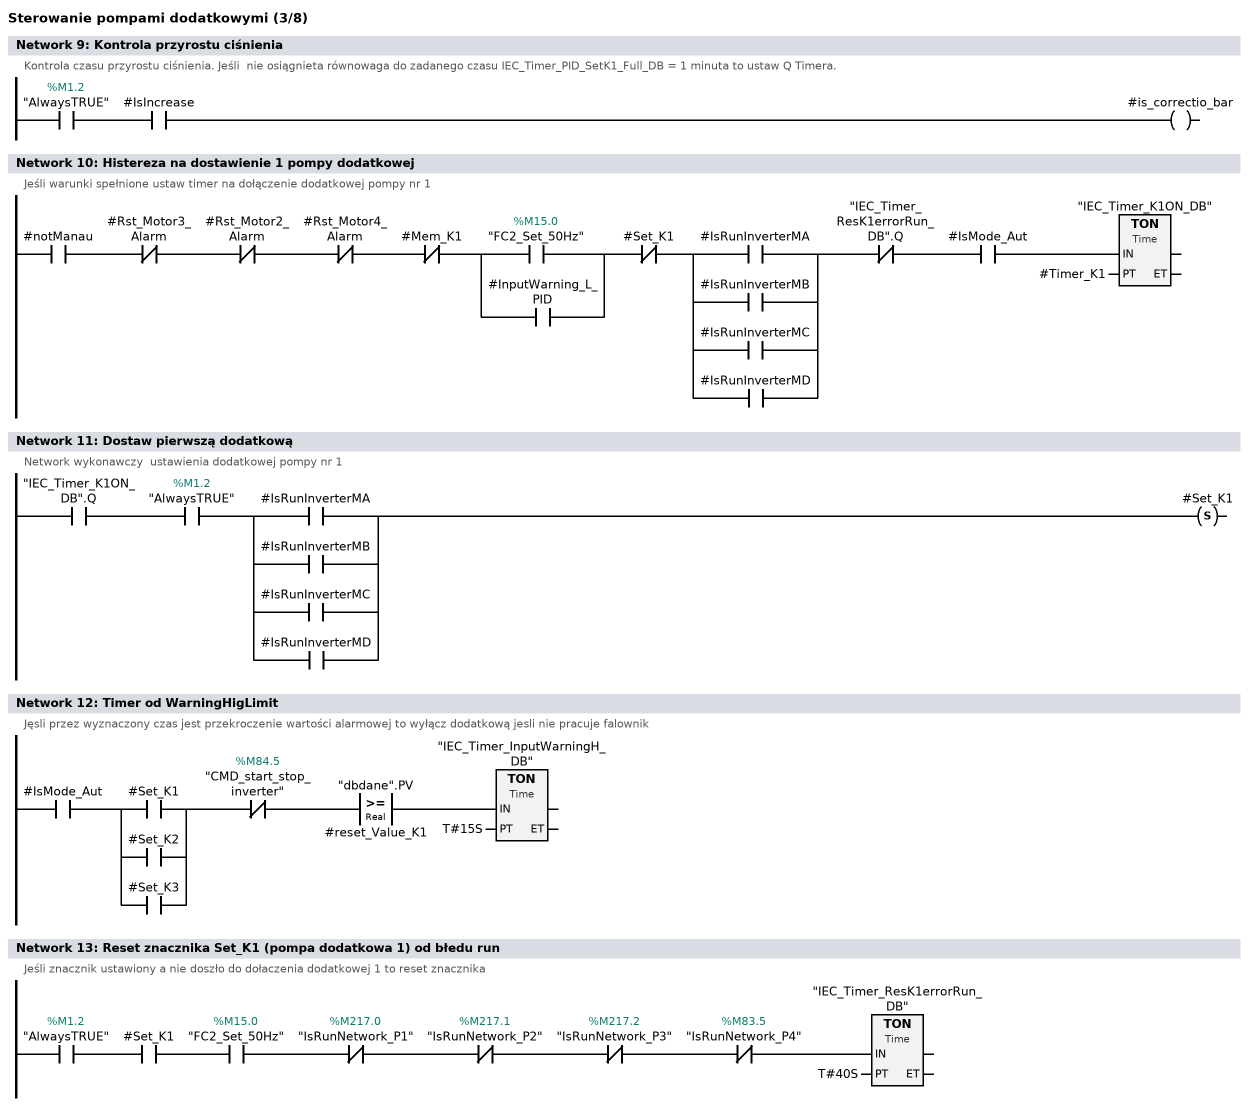
   RUNG wire#powerrail
      Contact( "AlwaysTRUE" )
      Contact( #IsIncrease )
      Coil( #is_correctio_bar )
   END_RUNG
   // the same network as SCL:
   #is_correctio_bar := "AlwaysTRUE" AND #IsIncrease;
END_REGION

REGION Network 10: Histereza na dostawienie 1 pompy dodatkowej
   // Jeśli warunki spełnione ustaw timer na dołączenie dodatkowej pompy nr 1
   RUNG wire#powerrail
      Contact( #notManau )
      I_Contact( #Rst_Motor3_Alarm )
      I_Contact( #Rst_Motor2_Alarm )
      I_Contact( #Rst_Motor4_Alarm )
      I_Contact( #Mem_K1 )
      wire#w1
      Contact( "FC2_Set_50Hz" )
      wire#w2
      I_Contact( #Set_K1 )
      wire#w3
      Contact( #IsRunInverterMA )
      wire#w4
      I_Contact( "IEC_Timer_ResK1errorRun_DB".Q )
      Contact( #IsMode_Aut )
      { S7_Templates := "time_type := Time" } "IEC_Timer_K1ON_DB".TON(pt := #Timer_K1, et =>)
   END_RUNG
   RUNG wire#w1
      Contact( #InputWarning_L_PID )
   END_RUNG wire#w2
   RUNG wire#w3
      Contact( #IsRunInverterMB )
   END_RUNG wire#w4
   RUNG wire#w3
      Contact( #IsRunInverterMC )
   END_RUNG wire#w4
   RUNG wire#w3
      Contact( #IsRunInverterMD )
   END_RUNG wire#w4
   // the same network as SCL:
   "IEC_Timer_K1ON_DB".TON(IN := #notManau AND NOT #Rst_Motor3_Alarm AND NOT #Rst_Motor2_Alarm AND NOT #Rst_Motor4_Alarm AND NOT #Mem_K1 AND ("FC2_Set_50Hz" OR #InputWarning_L_PID) AND NOT #Set_K1 AND (#IsRunInverterMA OR #IsRunInverterMB OR #IsRunInverterMC OR #IsRunInverterMD) AND NOT "IEC_Timer_ResK1errorRun_DB".Q AND #IsMode_Aut,
                           PT := #Timer_K1);
END_REGION

REGION Network 11: Dostaw pierwszą dodatkową
   // Network wykonawczy  ustawienia dodatkowej pompy nr 1
   RUNG wire#powerrail
      Contact( "IEC_Timer_K1ON_DB".Q )
      Contact( "AlwaysTRUE" )
      wire#w1
      Contact( #IsRunInverterMA )
      wire#w2
      S_Coil( #Set_K1 )
   END_RUNG
   RUNG wire#w1
      Contact( #IsRunInverterMB )
   END_RUNG wire#w2
   RUNG wire#w1
      Contact( #IsRunInverterMC )
   END_RUNG wire#w2
   RUNG wire#w1
      Contact( #IsRunInverterMD )
   END_RUNG wire#w2
   // the same network as SCL:
   IF "IEC_Timer_K1ON_DB".Q AND "AlwaysTRUE" AND (#IsRunInverterMA OR #IsRunInverterMB OR #IsRunInverterMC OR #IsRunInverterMD) THEN
       #Set_K1 := TRUE;
   END_IF;
END_REGION

REGION Network 12: Timer od WarningHigLimit
   // Jęsli przez wyznaczony czas jest przekroczenie wartości alarmowej to wyłącz dodatkową jesli nie pracuje falownik
   RUNG wire#powerrail
      Contact( #IsMode_Aut )
      wire#w1
      Contact( #Set_K1 )
      wire#w2
      I_Contact( "CMD_start_stop_inverter" )
      { S7_Templates := "SrcType := Real" } GE_Contact(in1 := "dbdane".PV, in2 := #reset_Value_K1)
      { S7_Templates := "time_type := Time" } "IEC_Timer_InputWarningH_DB".TON(pt := T#15S, et =>)
   END_RUNG
   RUNG wire#w1
      Contact( #Set_K2 )
   END_RUNG wire#w2
   RUNG wire#w1
      Contact( #Set_K3 )
   END_RUNG wire#w2
   // the same network as SCL:
   "IEC_Timer_InputWarningH_DB".TON(IN := #IsMode_Aut AND (#Set_K1 OR #Set_K2 OR #Set_K3) AND NOT "CMD_start_stop_inverter" AND ("dbdane".PV >= #reset_Value_K1),
                           PT := T#15S);
END_REGION

REGION Network 13: Reset znacznika Set_K1 (pompa dodatkowa 1) od błedu run
   // Jeśli znacznik ustawiony a nie doszło do dołaczenia dodatkowej 1 to reset znacznika
   RUNG wire#powerrail
      Contact( "AlwaysTRUE" )
      Contact( #Set_K1 )
      Contact( "FC2_Set_50Hz" )
      I_Contact( "IsRunNetwork_P1" )
      I_Contact( "IsRunNetwork_P2" )
      I_Contact( "IsRunNetwork_P3" )
      I_Contact( "IsRunNetwork_P4" )
      { S7_Templates := "time_type := Time" } "IEC_Timer_ResK1errorRun_DB".TON(pt := T#40S, et =>)
   END_RUNG
   // the same network as SCL:
   "IEC_Timer_ResK1errorRun_DB".TON(IN := "AlwaysTRUE" AND #Set_K1 AND "FC2_Set_50Hz" AND NOT "IsRunNetwork_P1" AND NOT "IsRunNetwork_P2" AND NOT "IsRunNetwork_P3" AND NOT "IsRunNetwork_P4",
                           PT := T#40S);
END_REGION

REGION Network 14: Flaga odłaczenia dodatkowej
   // Odłączenie gdy falownik wyłączony i alarm z PID WarningHi
   // Odłączenie gdy alarmowa ciśnienia
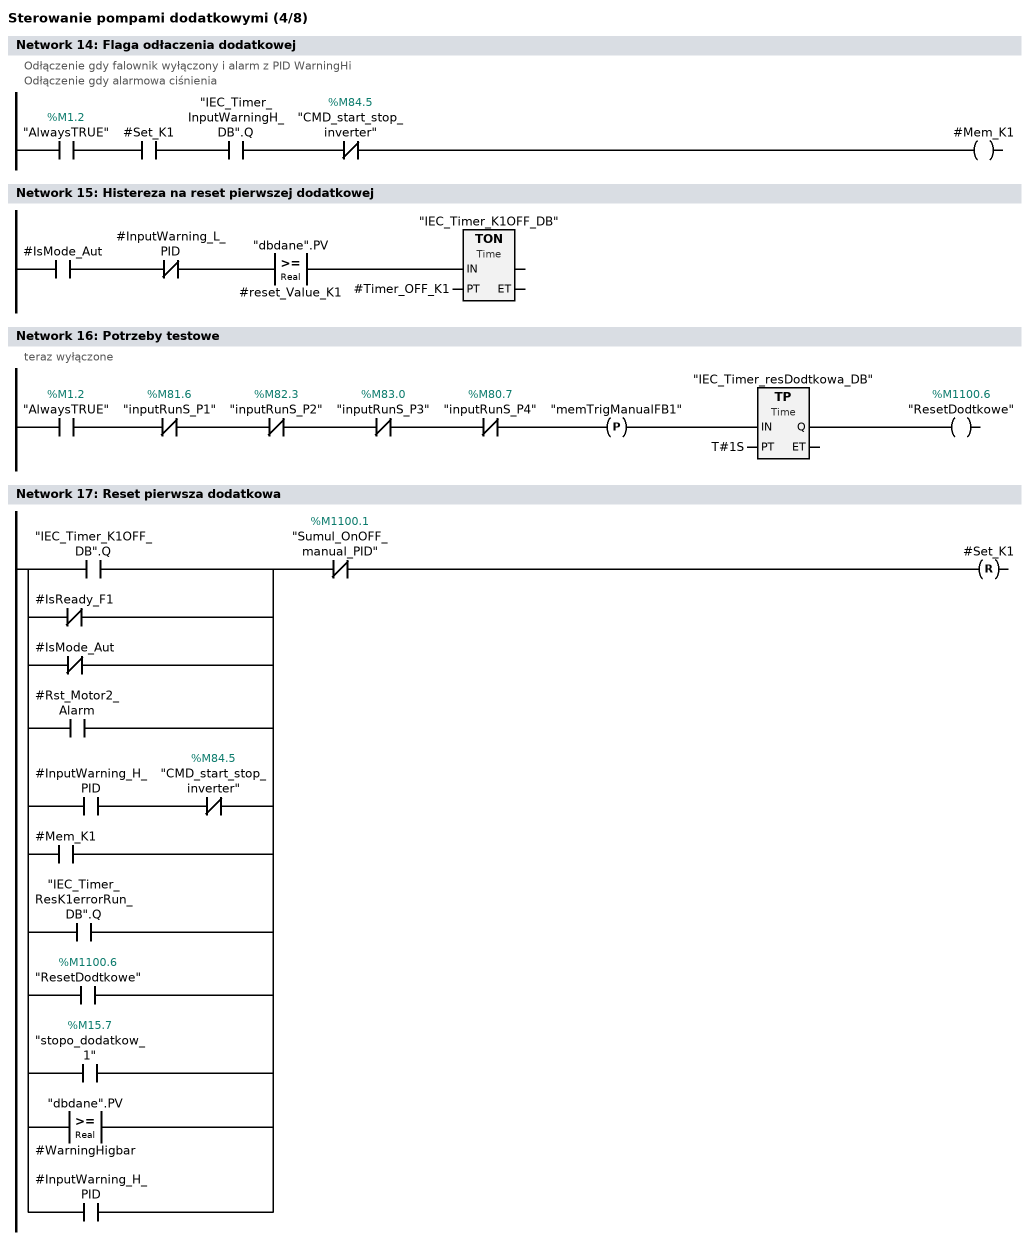
   RUNG wire#powerrail
      Contact( "AlwaysTRUE" )
      Contact( #Set_K1 )
      Contact( "IEC_Timer_InputWarningH_DB".Q )
      I_Contact( "CMD_start_stop_inverter" )
      Coil( #Mem_K1 )
   END_RUNG
   // the same network as SCL:
   #Mem_K1 := "AlwaysTRUE" AND #Set_K1 AND "IEC_Timer_InputWarningH_DB".Q AND NOT "CMD_start_stop_inverter";
END_REGION

REGION Network 15: Histereza na reset pierwszej dodatkowej
   RUNG wire#powerrail
      Contact( #IsMode_Aut )
      I_Contact( #InputWarning_L_PID )
      { S7_Templates := "SrcType := Real" } GE_Contact(in1 := "dbdane".PV, in2 := #reset_Value_K1)
      { S7_Templates := "time_type := Time" } "IEC_Timer_K1OFF_DB".TON(pt := #Timer_OFF_K1, et =>)
   END_RUNG
   // the same network as SCL:
   "IEC_Timer_K1OFF_DB".TON(IN := #IsMode_Aut AND NOT #InputWarning_L_PID AND ("dbdane".PV >= #reset_Value_K1),
                           PT := #Timer_OFF_K1);
END_REGION

REGION Network 16: Potrzeby testowe
   // teraz wyłączone
   RUNG wire#powerrail
      Contact( "AlwaysTRUE" )
      I_Contact( "inputRunS_P1" )
      I_Contact( "inputRunS_P2" )
      I_Contact( "inputRunS_P3" )
      I_Contact( "inputRunS_P4" )
      P_Trig( "memTrigManualFB1" )
      { S7_Templates := "time_type := Time" } "IEC_Timer_resDodtkowa_DB".TP(pt := T#1S, et =>)
      Coil( "ResetDodtkowe" )
   END_RUNG
   // the same network as SCL:
   #_w1 := "AlwaysTRUE" AND NOT "inputRunS_P1" AND NOT "inputRunS_P2" AND NOT "inputRunS_P3" AND NOT "inputRunS_P4";
   #_w2 := #_w1 AND NOT "memTrigManualFB1";   // rising edge
   "memTrigManualFB1" := #_w1;
   "IEC_Timer_resDodtkowa_DB".TP(IN := #_w2, PT := T#1S);
   "ResetDodtkowe" := "IEC_Timer_resDodtkowa_DB".Q;
END_REGION

REGION Network 17: Reset pierwsza dodatkowa
   RUNG wire#powerrail
      Contact( "IEC_Timer_K1OFF_DB".Q )
      wire#w1
      I_Contact( "Sumul_OnOFF_manual_PID" )
      R_Coil( #Set_K1 )
   END_RUNG
   RUNG wire#powerrail
      I_Contact( #IsReady_F1 )
   END_RUNG wire#w1
   RUNG wire#powerrail
      I_Contact( #IsMode_Aut )
   END_RUNG wire#w1
   RUNG wire#powerrail
      Contact( #Rst_Motor2_Alarm )
   END_RUNG wire#w1
   RUNG wire#powerrail
      Contact( #InputWarning_H_PID )
      I_Contact( "CMD_start_stop_inverter" )
   END_RUNG wire#w1
   RUNG wire#powerrail
      Contact( #Mem_K1 )
   END_RUNG wire#w1
   RUNG wire#powerrail
      Contact( "IEC_Timer_ResK1errorRun_DB".Q )
   END_RUNG wire#w1
   RUNG wire#powerrail
      Contact( "ResetDodtkowe" )
   END_RUNG wire#w1
   RUNG wire#powerrail
      Contact( "stopo_dodatkow_1" )
   END_RUNG wire#w1
   RUNG wire#powerrail
      { S7_Templates := "SrcType := Real" } GE_Contact(in1 := "dbdane".PV, in2 := #WarningHigbar)
   END_RUNG wire#w1
   RUNG wire#powerrail
      Contact( #InputWarning_H_PID )
   END_RUNG wire#w1
   // the same network as SCL:
   IF ("IEC_Timer_K1OFF_DB".Q OR NOT #IsReady_F1 OR NOT #IsMode_Aut OR #Rst_Motor2_Alarm OR (#InputWarning_H_PID AND NOT "CMD_start_stop_inverter") OR #Mem_K1 OR "IEC_Timer_ResK1errorRun_DB".Q OR "ResetDodtkowe" OR "stopo_dodatkow_1" OR ("dbdane".PV >= #WarningHigbar) OR #InputWarning_H_PID) AND NOT "Sumul_OnOFF_manual_PID" THEN
       #Set_K1 := FALSE;
   END_IF;
END_REGION

REGION Network 18: sterowanie wyłączeniem selektywnym dodatkowej 1
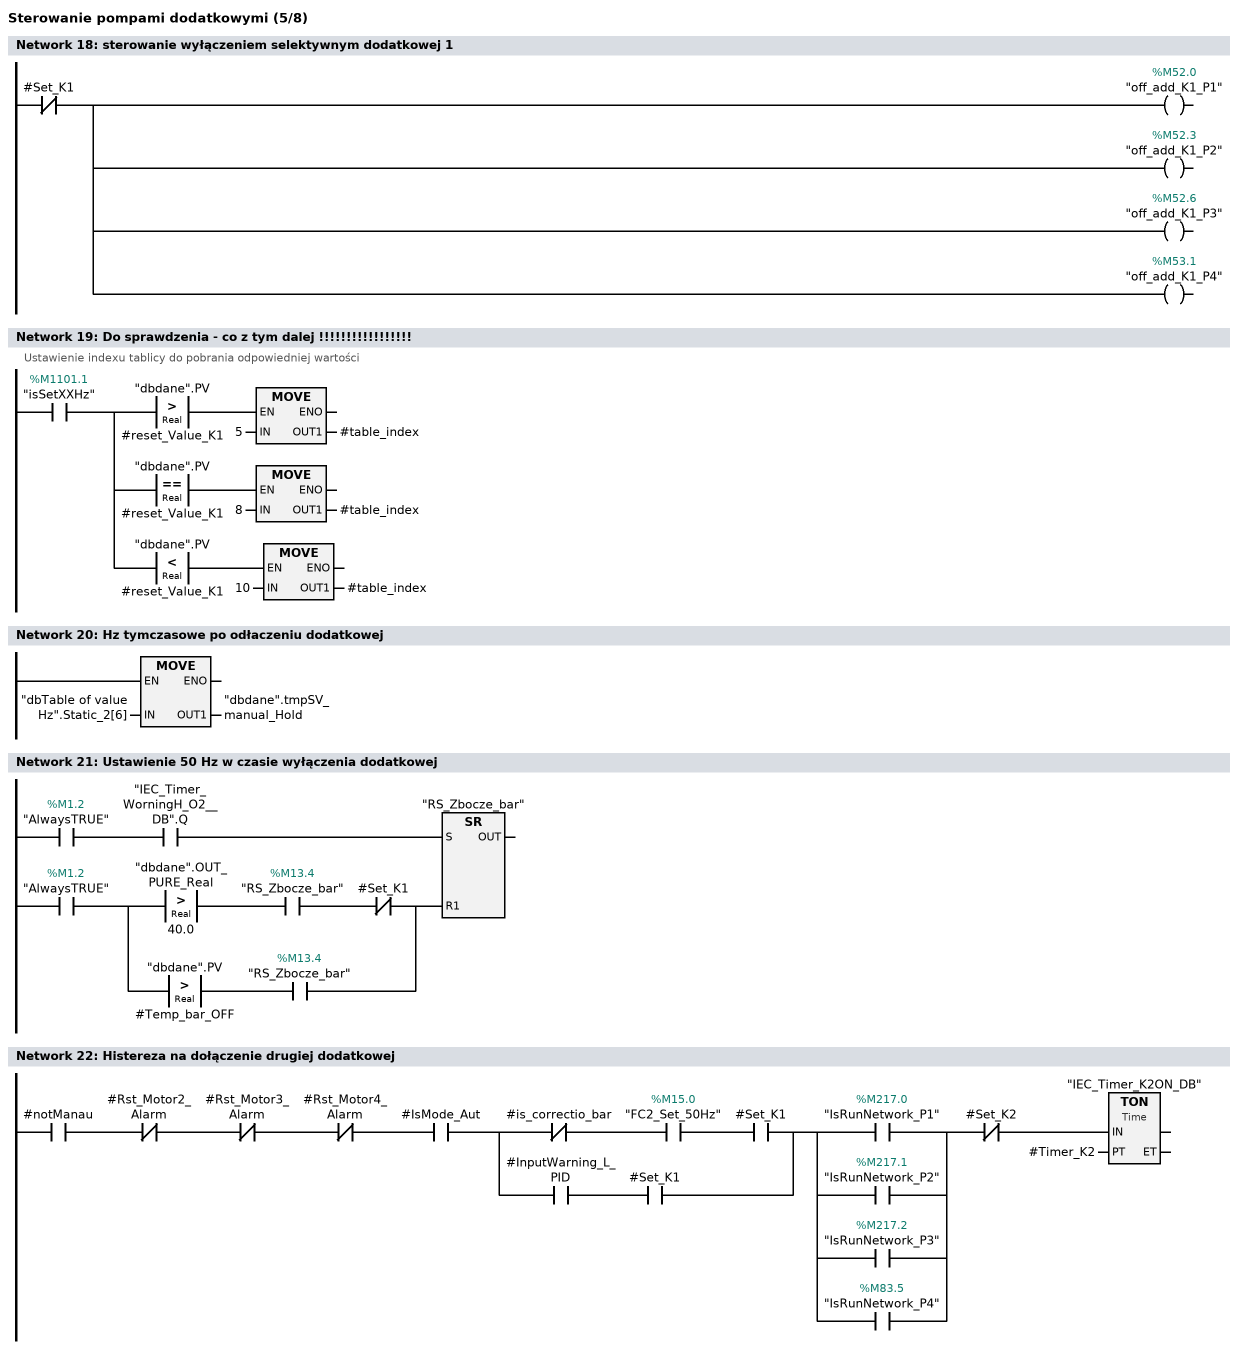
   RUNG wire#powerrail
      I_Contact( #Set_K1 )
      wire#w1
      Coil( "off_add_K1_P1" )
   END_RUNG
   RUNG wire#w1
      Coil( "off_add_K1_P2" )
   END_RUNG
   RUNG wire#w1
      Coil( "off_add_K1_P3" )
   END_RUNG
   RUNG wire#w1
      Coil( "off_add_K1_P4" )
   END_RUNG
   // the same network as SCL:
   "off_add_K1_P1" := NOT #Set_K1;
   "off_add_K1_P2" := NOT #Set_K1;
   "off_add_K1_P3" := NOT #Set_K1;
   "off_add_K1_P4" := NOT #Set_K1;
END_REGION

REGION Network 19: Do sprawdzenia - co z tym dalej !!!!!!!!!!!!!!!!!
   // Ustawienie indexu tablicy do pobrania odpowiedniej wartości
   RUNG wire#powerrail
      Contact( "isSetXXHz" )
      wire#w1
      { S7_Templates := "SrcType := Real" } GT_Contact(in1 := "dbdane".PV, in2 := #reset_Value_K1)
      Move(in := 5, out1 => #table_index)
   END_RUNG
   RUNG wire#w1
      { S7_Templates := "SrcType := Real" } EQ_Contact(in1 := "dbdane".PV, in2 := #reset_Value_K1)
      Move(in := 8, out1 => #table_index)
   END_RUNG
   RUNG wire#w1
      { S7_Templates := "SrcType := Real" } LT_Contact(in1 := "dbdane".PV, in2 := #reset_Value_K1)
      Move(in := 10, out1 => #table_index)
   END_RUNG
   // the same network as SCL:
   IF "isSetXXHz" AND ("dbdane".PV > #reset_Value_K1) THEN #table_index := 5; END_IF;
   IF "isSetXXHz" AND ("dbdane".PV = #reset_Value_K1) THEN #table_index := 8; END_IF;
   IF "isSetXXHz" AND ("dbdane".PV < #reset_Value_K1) THEN #table_index := 10; END_IF;
END_REGION

REGION Network 20: Hz tymczasowe po odłaczeniu dodatkowej
   RUNG wire#powerrail
      Move(in := "dbTable of value Hz".Static_2[6], out1 => "dbdane".tmpSV_manual_Hold)
   END_RUNG
   // the same network as SCL:
   "dbdane".tmpSV_manual_Hold := "dbTable of value Hz".Static_2[6];
END_REGION

REGION Network 21: Ustawienie 50 Hz w czasie wyłączenia dodatkowej
   RUNG wire#powerrail
      Contact( "AlwaysTRUE" )
      Contact( "IEC_Timer_WorningH_O2__DB".Q )
      S_SR(operand := "RS_Zbocze_bar", r1 := wire#w2)
   END_RUNG
   RUNG wire#powerrail
      Contact( "AlwaysTRUE" )
      wire#w1
      { S7_Templates := "SrcType := Real" } GT_Contact(in1 := "dbdane".OUT_PURE_Real, in2 := 40.0)
      Contact( "RS_Zbocze_bar" )
      I_Contact( #Set_K1 )
   END_RUNG wire#w2
   RUNG wire#w1
      { S7_Templates := "SrcType := Real" } GT_Contact(in1 := "dbdane".PV, in2 := #Temp_bar_OFF)
      Contact( "RS_Zbocze_bar" )
   END_RUNG wire#w2
   // the same network as SCL:
   #_w1 := "AlwaysTRUE" AND ((("dbdane".OUT_PURE_Real > 40.0) AND "RS_Zbocze_bar" AND NOT #Set_K1) OR (("dbdane".PV > #Temp_bar_OFF) AND "RS_Zbocze_bar"));
   IF "AlwaysTRUE" AND "IEC_Timer_WorningH_O2__DB".Q THEN
       "RS_Zbocze_bar" := TRUE;   // SR flip-flop
   END_IF;
   IF #_w1 THEN "RS_Zbocze_bar" := FALSE; END_IF;
END_REGION

REGION Network 22: Histereza na dołączenie drugiej dodatkowej
   RUNG wire#powerrail
      Contact( #notManau )
      I_Contact( #Rst_Motor2_Alarm )
      I_Contact( #Rst_Motor3_Alarm )
      I_Contact( #Rst_Motor4_Alarm )
      Contact( #IsMode_Aut )
      wire#w1
      I_Contact( #is_correctio_bar )
      Contact( "FC2_Set_50Hz" )
      Contact( #Set_K1 )
      wire#w2
      Contact( "IsRunNetwork_P1" )
      wire#w3
      I_Contact( #Set_K2 )
      { S7_Templates := "time_type := Time" } "IEC_Timer_K2ON_DB".TON(pt := #Timer_K2, et =>)
   END_RUNG
   RUNG wire#w1
      Contact( #InputWarning_L_PID )
      Contact( #Set_K1 )
   END_RUNG wire#w2
   RUNG wire#w2
      Contact( "IsRunNetwork_P2" )
   END_RUNG wire#w3
   RUNG wire#w2
      Contact( "IsRunNetwork_P3" )
   END_RUNG wire#w3
   RUNG wire#w2
      Contact( "IsRunNetwork_P4" )
   END_RUNG wire#w3
   // the same network as SCL:
   "IEC_Timer_K2ON_DB".TON(IN := #notManau AND NOT #Rst_Motor2_Alarm AND NOT #Rst_Motor3_Alarm AND NOT #Rst_Motor4_Alarm AND #IsMode_Aut AND ((NOT #is_correctio_bar AND "FC2_Set_50Hz" AND #Set_K1) OR (#InputWarning_L_PID AND #Set_K1)) AND ("IsRunNetwork_P1" OR "IsRunNetwork_P2" OR "IsRunNetwork_P3" OR "IsRunNetwork_P4") AND NOT #Set_K2,
                           PT := #Timer_K2);
END_REGION

REGION Network 23: Dostawienie drugiej dodatkowej
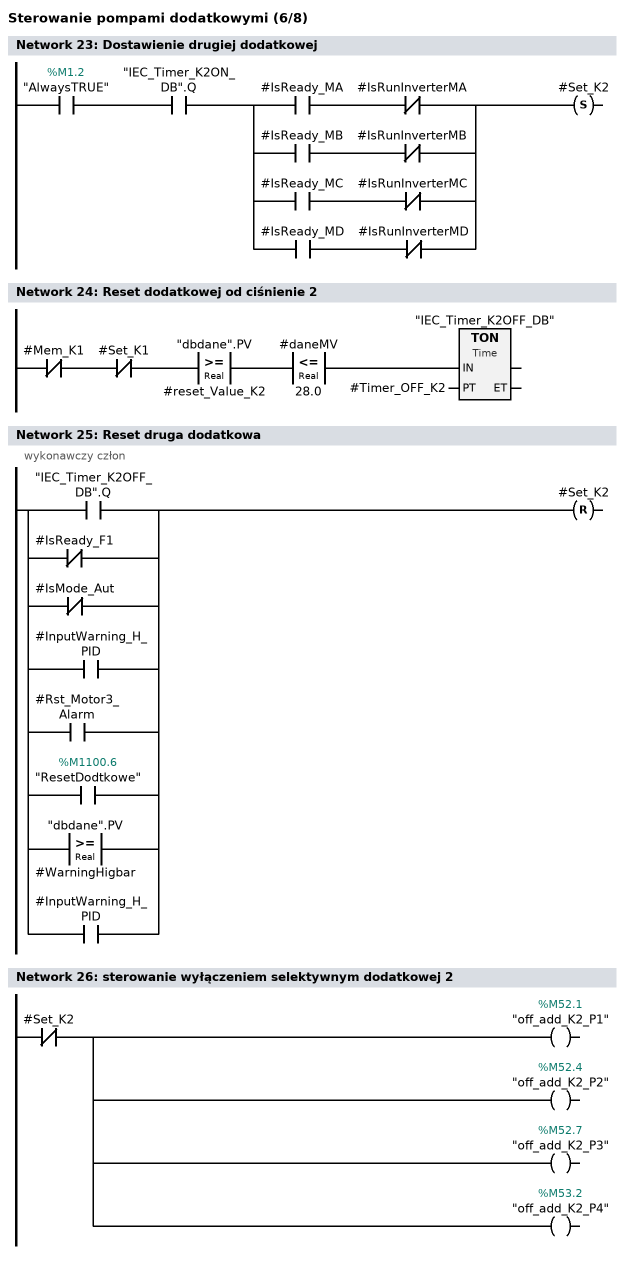
   RUNG wire#powerrail
      Contact( "AlwaysTRUE" )
      Contact( "IEC_Timer_K2ON_DB".Q )
      wire#w1
      Contact( #IsReady_MA )
      I_Contact( #IsRunInverterMA )
      wire#w2
      S_Coil( #Set_K2 )
   END_RUNG
   RUNG wire#w1
      Contact( #IsReady_MB )
      I_Contact( #IsRunInverterMB )
   END_RUNG wire#w2
   RUNG wire#w1
      Contact( #IsReady_MC )
      I_Contact( #IsRunInverterMC )
   END_RUNG wire#w2
   RUNG wire#w1
      Contact( #IsReady_MD )
      I_Contact( #IsRunInverterMD )
   END_RUNG wire#w2
   // the same network as SCL:
   IF "AlwaysTRUE" AND "IEC_Timer_K2ON_DB".Q AND ((#IsReady_MA AND NOT #IsRunInverterMA) OR (#IsReady_MB AND NOT #IsRunInverterMB) OR (#IsReady_MC AND NOT #IsRunInverterMC) OR (#IsReady_MD AND NOT #IsRunInverterMD)) THEN
       #Set_K2 := TRUE;
   END_IF;
END_REGION

REGION Network 24: Reset dodatkowej od ciśnienie 2
   RUNG wire#powerrail
      I_Contact( #Mem_K1 )
      I_Contact( #Set_K1 )
      { S7_Templates := "SrcType := Real" } GE_Contact(in1 := "dbdane".PV, in2 := #reset_Value_K2)
      { S7_Templates := "SrcType := Real" } LE_Contact(in1 := #daneMV, in2 := 28.0)
      { S7_Templates := "time_type := Time" } "IEC_Timer_K2OFF_DB".TON(pt := #Timer_OFF_K2, et =>)
   END_RUNG
   // the same network as SCL:
   "IEC_Timer_K2OFF_DB".TON(IN := NOT #Mem_K1 AND NOT #Set_K1 AND ("dbdane".PV >= #reset_Value_K2) AND (#daneMV <= 28.0),
                           PT := #Timer_OFF_K2);
END_REGION

REGION Network 25: Reset druga dodatkowa
   // wykonawczy człon
   RUNG wire#powerrail
      Contact( "IEC_Timer_K2OFF_DB".Q )
      wire#w1
      R_Coil( #Set_K2 )
   END_RUNG
   RUNG wire#powerrail
      I_Contact( #IsReady_F1 )
   END_RUNG wire#w1
   RUNG wire#powerrail
      I_Contact( #IsMode_Aut )
   END_RUNG wire#w1
   RUNG wire#powerrail
      Contact( #InputWarning_H_PID )
   END_RUNG wire#w1
   RUNG wire#powerrail
      Contact( #Rst_Motor3_Alarm )
   END_RUNG wire#w1
   RUNG wire#powerrail
      Contact( "ResetDodtkowe" )
   END_RUNG wire#w1
   RUNG wire#powerrail
      { S7_Templates := "SrcType := Real" } GE_Contact(in1 := "dbdane".PV, in2 := #WarningHigbar)
   END_RUNG wire#w1
   RUNG wire#powerrail
      Contact( #InputWarning_H_PID )
   END_RUNG wire#w1
   // the same network as SCL:
   IF "IEC_Timer_K2OFF_DB".Q OR NOT #IsReady_F1 OR NOT #IsMode_Aut OR #InputWarning_H_PID OR #Rst_Motor3_Alarm OR "ResetDodtkowe" OR ("dbdane".PV >= #WarningHigbar) OR #InputWarning_H_PID THEN
       #Set_K2 := FALSE;
   END_IF;
END_REGION

REGION Network 26: sterowanie wyłączeniem selektywnym dodatkowej 2
   RUNG wire#powerrail
      I_Contact( #Set_K2 )
      wire#w1
      Coil( "off_add_K2_P1" )
   END_RUNG
   RUNG wire#w1
      Coil( "off_add_K2_P2" )
   END_RUNG
   RUNG wire#w1
      Coil( "off_add_K2_P3" )
   END_RUNG
   RUNG wire#w1
      Coil( "off_add_K2_P4" )
   END_RUNG
   // the same network as SCL:
   "off_add_K2_P1" := NOT #Set_K2;
   "off_add_K2_P2" := NOT #Set_K2;
   "off_add_K2_P3" := NOT #Set_K2;
   "off_add_K2_P4" := NOT #Set_K2;
END_REGION

REGION Network 27: Trzecia dodatkowa dołączenie
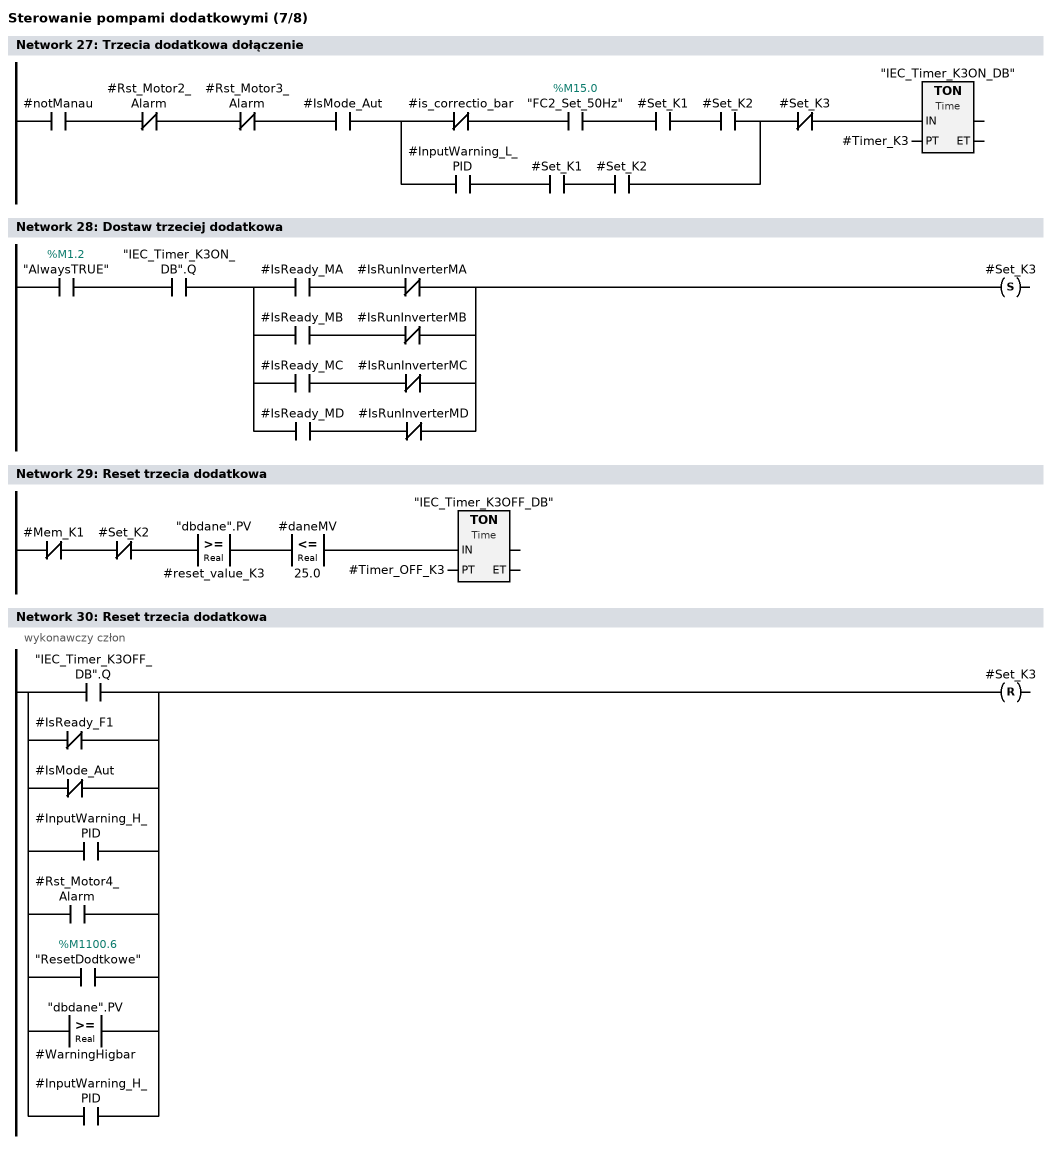
   RUNG wire#powerrail
      Contact( #notManau )
      I_Contact( #Rst_Motor2_Alarm )
      I_Contact( #Rst_Motor3_Alarm )
      Contact( #IsMode_Aut )
      wire#w1
      I_Contact( #is_correctio_bar )
      Contact( "FC2_Set_50Hz" )
      Contact( #Set_K1 )
      Contact( #Set_K2 )
      wire#w2
      I_Contact( #Set_K3 )
      { S7_Templates := "time_type := Time" } "IEC_Timer_K3ON_DB".TON(pt := #Timer_K3, et =>)
   END_RUNG
   RUNG wire#w1
      Contact( #InputWarning_L_PID )
      Contact( #Set_K1 )
      Contact( #Set_K2 )
   END_RUNG wire#w2
   // the same network as SCL:
   "IEC_Timer_K3ON_DB".TON(IN := #notManau AND NOT #Rst_Motor2_Alarm AND NOT #Rst_Motor3_Alarm AND #IsMode_Aut AND ((NOT #is_correctio_bar AND "FC2_Set_50Hz" AND #Set_K1 AND #Set_K2) OR (#InputWarning_L_PID AND #Set_K1 AND #Set_K2)) AND NOT #Set_K3,
                           PT := #Timer_K3);
END_REGION

REGION Network 28: Dostaw trzeciej dodatkowa
   RUNG wire#powerrail
      Contact( "AlwaysTRUE" )
      Contact( "IEC_Timer_K3ON_DB".Q )
      wire#w1
      Contact( #IsReady_MA )
      I_Contact( #IsRunInverterMA )
      wire#w2
      S_Coil( #Set_K3 )
   END_RUNG
   RUNG wire#w1
      Contact( #IsReady_MB )
      I_Contact( #IsRunInverterMB )
   END_RUNG wire#w2
   RUNG wire#w1
      Contact( #IsReady_MC )
      I_Contact( #IsRunInverterMC )
   END_RUNG wire#w2
   RUNG wire#w1
      Contact( #IsReady_MD )
      I_Contact( #IsRunInverterMD )
   END_RUNG wire#w2
   // the same network as SCL:
   IF "AlwaysTRUE" AND "IEC_Timer_K3ON_DB".Q AND ((#IsReady_MA AND NOT #IsRunInverterMA) OR (#IsReady_MB AND NOT #IsRunInverterMB) OR (#IsReady_MC AND NOT #IsRunInverterMC) OR (#IsReady_MD AND NOT #IsRunInverterMD)) THEN
       #Set_K3 := TRUE;
   END_IF;
END_REGION

REGION Network 29: Reset trzecia dodatkowa
   RUNG wire#powerrail
      I_Contact( #Mem_K1 )
      I_Contact( #Set_K2 )
      { S7_Templates := "SrcType := Real" } GE_Contact(in1 := "dbdane".PV, in2 := #reset_value_K3)
      { S7_Templates := "SrcType := Real" } LE_Contact(in1 := #daneMV, in2 := 25.0)
      { S7_Templates := "time_type := Time" } "IEC_Timer_K3OFF_DB".TON(pt := #Timer_OFF_K3, et =>)
   END_RUNG
   // the same network as SCL:
   "IEC_Timer_K3OFF_DB".TON(IN := NOT #Mem_K1 AND NOT #Set_K2 AND ("dbdane".PV >= #reset_value_K3) AND (#daneMV <= 25.0),
                           PT := #Timer_OFF_K3);
END_REGION

REGION Network 30: Reset trzecia dodatkowa
   // wykonawczy człon
   RUNG wire#powerrail
      Contact( "IEC_Timer_K3OFF_DB".Q )
      wire#w1
      R_Coil( #Set_K3 )
   END_RUNG
   RUNG wire#powerrail
      I_Contact( #IsReady_F1 )
   END_RUNG wire#w1
   RUNG wire#powerrail
      I_Contact( #IsMode_Aut )
   END_RUNG wire#w1
   RUNG wire#powerrail
      Contact( #InputWarning_H_PID )
   END_RUNG wire#w1
   RUNG wire#powerrail
      Contact( #Rst_Motor4_Alarm )
   END_RUNG wire#w1
   RUNG wire#powerrail
      Contact( "ResetDodtkowe" )
   END_RUNG wire#w1
   RUNG wire#powerrail
      { S7_Templates := "SrcType := Real" } GE_Contact(in1 := "dbdane".PV, in2 := #WarningHigbar)
   END_RUNG wire#w1
   RUNG wire#powerrail
      Contact( #InputWarning_H_PID )
   END_RUNG wire#w1
   // the same network as SCL:
   IF "IEC_Timer_K3OFF_DB".Q OR NOT #IsReady_F1 OR NOT #IsMode_Aut OR #InputWarning_H_PID OR #Rst_Motor4_Alarm OR "ResetDodtkowe" OR ("dbdane".PV >= #WarningHigbar) OR #InputWarning_H_PID THEN
       #Set_K3 := FALSE;
   END_IF;
END_REGION

REGION Network 31: sterowanie wyłączeniem selektywnym dodatkowej 3
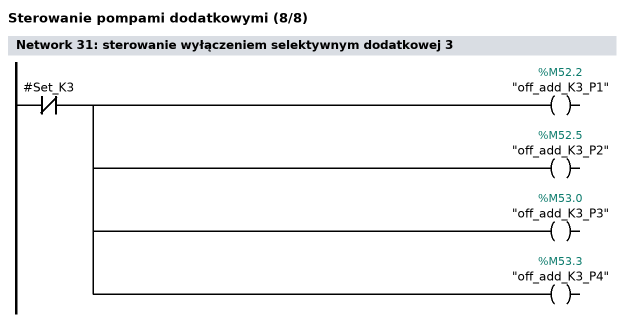
   RUNG wire#powerrail
      I_Contact( #Set_K3 )
      wire#w1
      Coil( "off_add_K3_P1" )
   END_RUNG
   RUNG wire#w1
      Coil( "off_add_K3_P2" )
   END_RUNG
   RUNG wire#w1
      Coil( "off_add_K3_P3" )
   END_RUNG
   RUNG wire#w1
      Coil( "off_add_K3_P4" )
   END_RUNG
   // the same network as SCL:
   "off_add_K3_P1" := NOT #Set_K3;
   "off_add_K3_P2" := NOT #Set_K3;
   "off_add_K3_P3" := NOT #Set_K3;
   "off_add_K3_P4" := NOT #Set_K3;
END_REGION
END_FUNCTION_BLOCK

FUNCTION_BLOCK "Ustawienie pomp wiodącej i dodatkowych"   // FB9, LAD
TITLE = Funkcja ustalająca napęd wiodący i dodatkowe
{ S7_Optimized_Access := 'TRUE' }
AUTHOR : rtecmer
VERSION : 0.1
// Ustalanie silnika wiodącego i dodatkowego następuje po sprawdzeniu czy dany napęd załączony jes na falownik czy na sieć. Procedura rozpoczyna się od ustalenia napedu wiodącego. / Ustalanie silnika wiodącego i dodatkowego następuje po sprawdzeniu czy dany napęd załączony jes na falownik czy na sieć. Procedura rozpoczyna się od ustalenia napędu wiodącego.
// stored: AutoNumber true, IsIECCheckEnabled false, IsRetainMemResEnabled false, MemoryReserve 500, SetENOAutomatically false, UDAEnableTagReadback false
   VAR_IN_OUT
      set_Motor2 : Bool;   // pomocniczy bit ustawiania pompę dodatkową nr1
      set_Motor3 : Bool;   // pomocniczy bit ustawiania pompę dodatkową nr2
      set_Motor4 : Bool;   // pomocniczy bit ustawiania pompę dodatkową nr3
   END_VAR
   VAR_TEMP
      tmp_Res_Motor2 : Bool;   // pomocniczy bit kasowania znacznika dodatkowej nr1
      tmp_Res_Motor3 : Bool;   // pomocniczy bit kasowania znacznika dodatkowej nr2
      tmp_Res_Motor4 : Bool;   // pomocniczy bit kasowania znacznika dodatkowej nr3
   END_VAR
   VAR_TEMP   // added for the SCL form of the ladder/FBD networks
      _w1 : Bool;
      _w2 : Bool;
      _w3 : Bool;
      _w4 : Bool;
      _w5 : Bool;
      _w6 : Bool;
   END_VAR
BEGIN

REGION Network 1: Znacznikdmuchawę wiodącej / Znacznik pompy wiodącej
   // M218.0 - bit ustalający pompę wiodącą . Przekazywany do zmiennych "IN" funkcji  "Control of   Inverters" napędów P1,P2,P3,P4 / M218.0 - bit ustalający pompy wiodącą . Przekazywany do zmiennych "IN" funkcji  "Control of   Inverters"
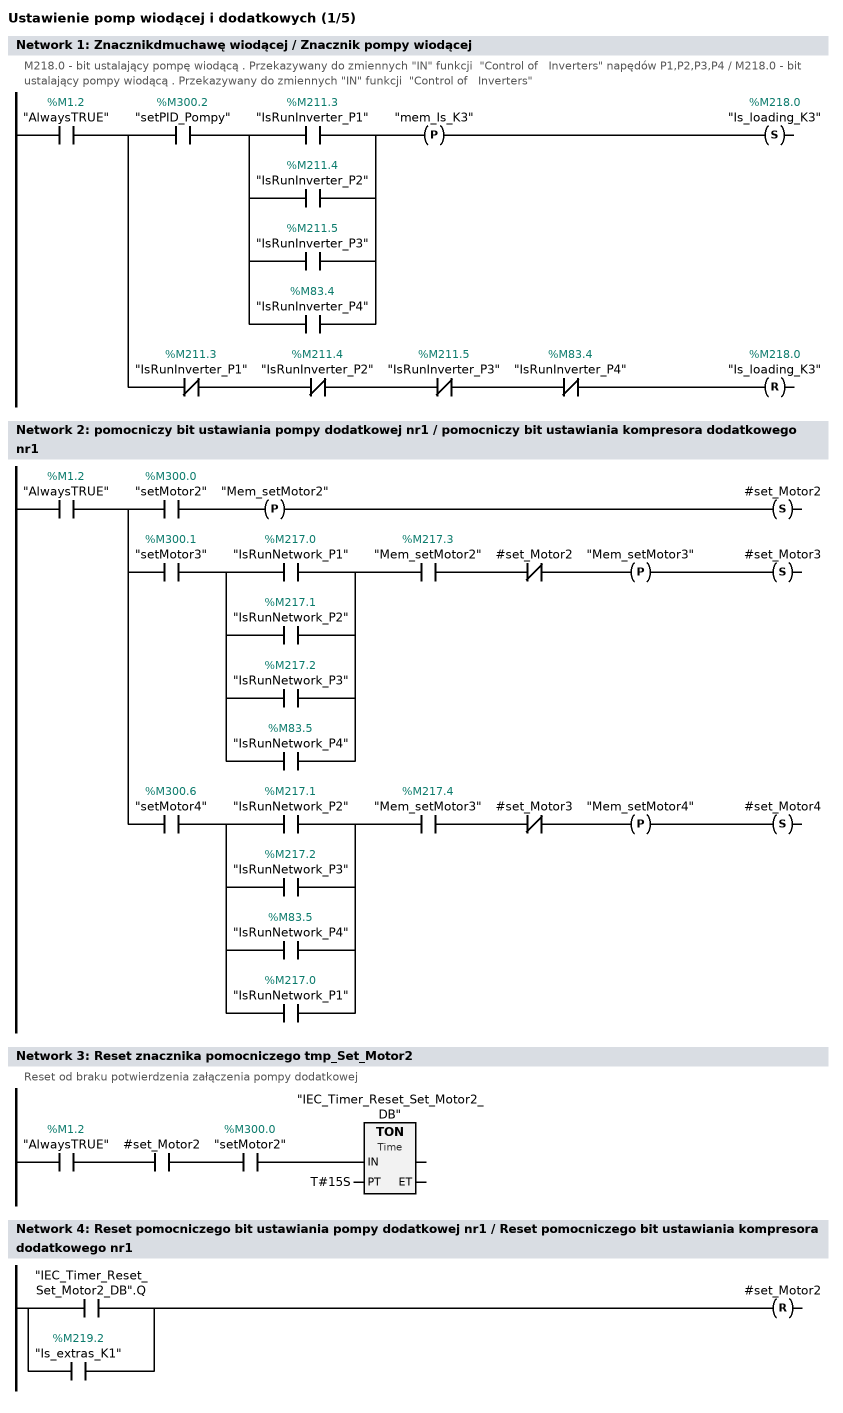
   RUNG wire#powerrail
      Contact( "AlwaysTRUE" )
      wire#w1
      Contact( "setPID_Pompy" )
      wire#w2
      Contact( "IsRunInverter_P1" )
      wire#w3
      P_Trig( "mem_Is_K3" )
      S_Coil( "Is_loading_K3" )
   END_RUNG
   RUNG wire#w2
      Contact( "IsRunInverter_P2" )
   END_RUNG wire#w3
   RUNG wire#w2
      Contact( "IsRunInverter_P3" )
   END_RUNG wire#w3
   RUNG wire#w2
      Contact( "IsRunInverter_P4" )
   END_RUNG wire#w3
   RUNG wire#w1
      I_Contact( "IsRunInverter_P1" )
      I_Contact( "IsRunInverter_P2" )
      I_Contact( "IsRunInverter_P3" )
      I_Contact( "IsRunInverter_P4" )
      R_Coil( "Is_loading_K3" )
   END_RUNG
   // the same network as SCL:
   #_w1 := "AlwaysTRUE" AND "setPID_Pompy" AND ("IsRunInverter_P1" OR "IsRunInverter_P2" OR "IsRunInverter_P3" OR "IsRunInverter_P4");
   #_w2 := #_w1 AND NOT "mem_Is_K3";   // rising edge
   "mem_Is_K3" := #_w1;
   IF #_w2 THEN "Is_loading_K3" := TRUE; END_IF;
   IF "AlwaysTRUE" AND NOT "IsRunInverter_P1" AND NOT "IsRunInverter_P2" AND NOT "IsRunInverter_P3" AND NOT "IsRunInverter_P4" THEN
       "Is_loading_K3" := FALSE;
   END_IF;
END_REGION

REGION Network 2: pomocniczy bit ustawiania pompy dodatkowej nr1 / pomocniczy bit ustawiania kompresora dodatkowego nr1
   RUNG wire#powerrail
      Contact( "AlwaysTRUE" )
      wire#w1
      Contact( "setMotor2" )
      P_Trig( "Mem_setMotor2" )
      S_Coil( #set_Motor2 )
   END_RUNG
   RUNG wire#w1
      Contact( "setMotor3" )
      wire#w2
      Contact( "IsRunNetwork_P1" )
      wire#w3
      Contact( "Mem_setMotor2" )
      I_Contact( #set_Motor2 )
      P_Trig( "Mem_setMotor3" )
      S_Coil( #set_Motor3 )
   END_RUNG
   RUNG wire#w2
      Contact( "IsRunNetwork_P2" )
   END_RUNG wire#w3
   RUNG wire#w2
      Contact( "IsRunNetwork_P3" )
   END_RUNG wire#w3
   RUNG wire#w2
      Contact( "IsRunNetwork_P4" )
   END_RUNG wire#w3
   RUNG wire#w1
      Contact( "setMotor4" )
      wire#w4
      Contact( "IsRunNetwork_P2" )
      wire#w5
      Contact( "Mem_setMotor3" )
      I_Contact( #set_Motor3 )
      P_Trig( "Mem_setMotor4" )
      S_Coil( #set_Motor4 )
   END_RUNG
   RUNG wire#w4
      Contact( "IsRunNetwork_P3" )
   END_RUNG wire#w5
   RUNG wire#w4
      Contact( "IsRunNetwork_P4" )
   END_RUNG wire#w5
   RUNG wire#w4
      Contact( "IsRunNetwork_P1" )
   END_RUNG wire#w5
   // the same network as SCL:
   #_w1 := "AlwaysTRUE" AND "setMotor2";
   #_w2 := #_w1 AND NOT "Mem_setMotor2";   // rising edge
   "Mem_setMotor2" := #_w1;
   IF #_w2 THEN #set_Motor2 := TRUE; END_IF;
   #_w3 := "AlwaysTRUE" AND "setMotor3" AND ("IsRunNetwork_P1" OR "IsRunNetwork_P2" OR "IsRunNetwork_P3" OR "IsRunNetwork_P4") AND "Mem_setMotor2" AND NOT #set_Motor2;
   #_w4 := #_w3 AND NOT "Mem_setMotor3";   // rising edge
   "Mem_setMotor3" := #_w3;
   IF #_w4 THEN #set_Motor3 := TRUE; END_IF;
   #_w5 := "AlwaysTRUE" AND "setMotor4" AND ("IsRunNetwork_P2" OR "IsRunNetwork_P3" OR "IsRunNetwork_P4" OR "IsRunNetwork_P1") AND "Mem_setMotor3" AND NOT #set_Motor3;
   #_w6 := #_w5 AND NOT "Mem_setMotor4";   // rising edge
   "Mem_setMotor4" := #_w5;
   IF #_w6 THEN #set_Motor4 := TRUE; END_IF;
END_REGION

REGION Network 3: Reset znacznika pomocniczego tmp_Set_Motor2
   // Reset od braku potwierdzenia załączenia pompy dodatkowej
   RUNG wire#powerrail
      Contact( "AlwaysTRUE" )
      Contact( #set_Motor2 )
      Contact( "setMotor2" )
      { S7_Templates := "time_type := Time" } "IEC_Timer_Reset_Set_Motor2_DB".TON(pt := T#15S, et =>)
   END_RUNG
   // the same network as SCL:
   "IEC_Timer_Reset_Set_Motor2_DB".TON(IN := "AlwaysTRUE" AND #set_Motor2 AND "setMotor2", PT := T#15S);
END_REGION

REGION Network 4: Reset pomocniczego bit ustawiania pompy dodatkowej nr1 / Reset pomocniczego bit ustawiania kompresora dodatkowego nr1
   RUNG wire#powerrail
      Contact( "IEC_Timer_Reset_Set_Motor2_DB".Q )
      wire#w1
      R_Coil( #set_Motor2 )
   END_RUNG
   RUNG wire#powerrail
      Contact( "Is_extras_K1" )
   END_RUNG wire#w1
   // the same network as SCL:
   IF "IEC_Timer_Reset_Set_Motor2_DB".Q OR "Is_extras_K1" THEN #set_Motor2 := FALSE; END_IF;
END_REGION

REGION Network 5: Reset znacznika pomocniczego tmp_Set_Motor3
   // Reset od braku potwierdzenia załączenia pompy dodatkowej / Reset od braku potwierdzenia załączenia pompy  dodatkowej
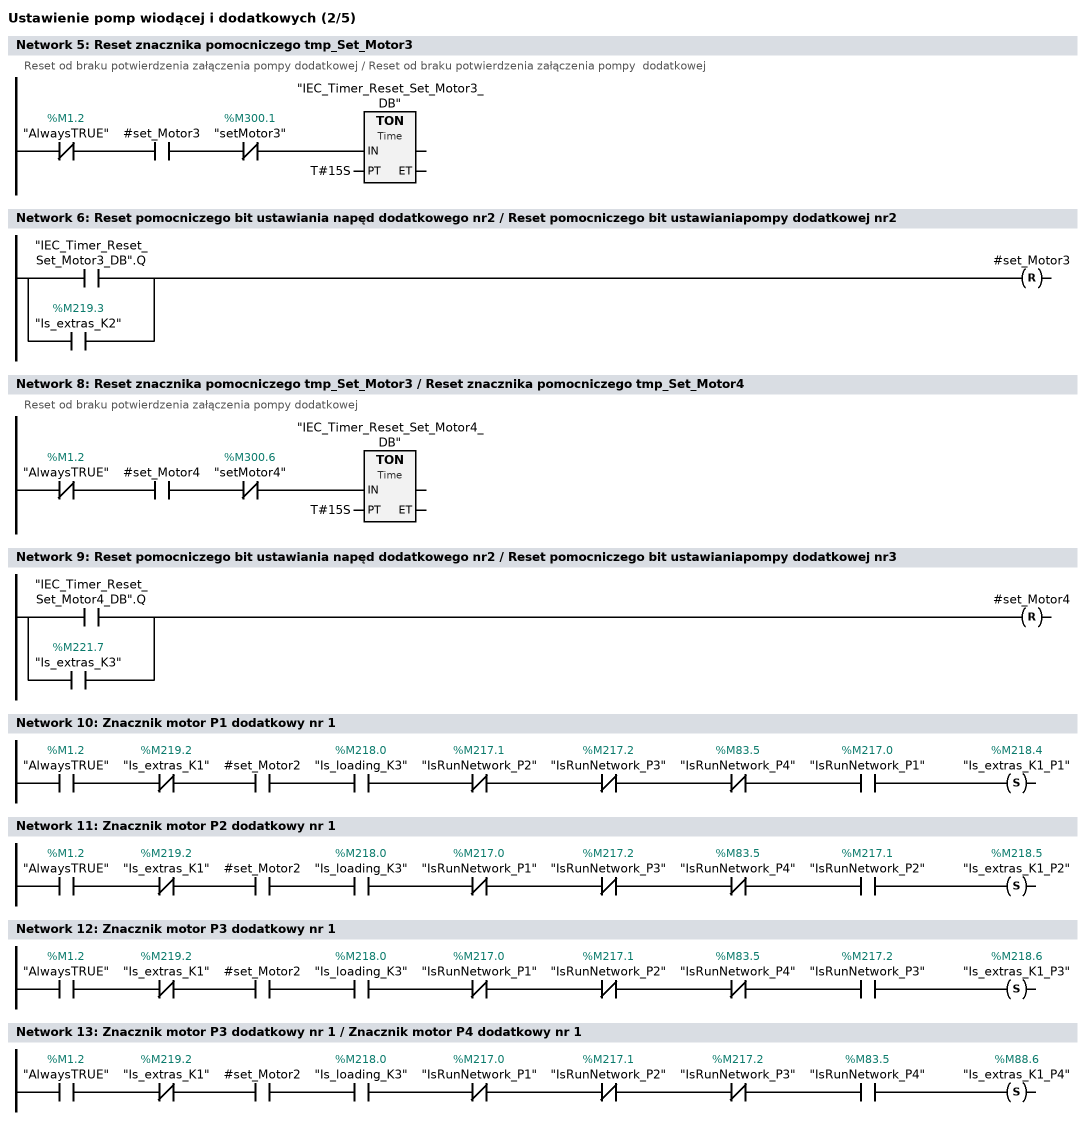
   RUNG wire#powerrail
      I_Contact( "AlwaysTRUE" )
      Contact( #set_Motor3 )
      I_Contact( "setMotor3" )
      { S7_Templates := "time_type := Time" } "IEC_Timer_Reset_Set_Motor3_DB".TON(pt := T#15S, et =>)
   END_RUNG
   // the same network as SCL:
   "IEC_Timer_Reset_Set_Motor3_DB".TON(IN := NOT "AlwaysTRUE" AND #set_Motor3 AND NOT "setMotor3", PT := T#15S);
END_REGION

REGION Network 6: Reset pomocniczego bit ustawiania napęd dodatkowego nr2 / Reset pomocniczego bit ustawianiapompy dodatkowej nr2
   RUNG wire#powerrail
      Contact( "IEC_Timer_Reset_Set_Motor3_DB".Q )
      wire#w1
      R_Coil( #set_Motor3 )
   END_RUNG
   RUNG wire#powerrail
      Contact( "Is_extras_K2" )
   END_RUNG wire#w1
   // the same network as SCL:
   IF "IEC_Timer_Reset_Set_Motor3_DB".Q OR "Is_extras_K2" THEN #set_Motor3 := FALSE; END_IF;
END_REGION

REGION Network 8: Reset znacznika pomocniczego tmp_Set_Motor3 / Reset znacznika pomocniczego tmp_Set_Motor4
   // Reset od braku potwierdzenia załączenia pompy dodatkowej
   RUNG wire#powerrail
      I_Contact( "AlwaysTRUE" )
      Contact( #set_Motor4 )
      I_Contact( "setMotor4" )
      { S7_Templates := "time_type := Time" } "IEC_Timer_Reset_Set_Motor4_DB".TON(pt := T#15S, et =>)
   END_RUNG
   // the same network as SCL:
   "IEC_Timer_Reset_Set_Motor4_DB".TON(IN := NOT "AlwaysTRUE" AND #set_Motor4 AND NOT "setMotor4", PT := T#15S);
END_REGION

REGION Network 9: Reset pomocniczego bit ustawiania napęd dodatkowego nr2 / Reset pomocniczego bit ustawianiapompy dodatkowej nr3
   RUNG wire#powerrail
      Contact( "IEC_Timer_Reset_Set_Motor4_DB".Q )
      wire#w1
      R_Coil( #set_Motor4 )
   END_RUNG
   RUNG wire#powerrail
      Contact( "Is_extras_K3" )
   END_RUNG wire#w1
   // the same network as SCL:
   IF "IEC_Timer_Reset_Set_Motor4_DB".Q OR "Is_extras_K3" THEN #set_Motor4 := FALSE; END_IF;
END_REGION

REGION Network 10: Znacznik motor P1 dodatkowy nr 1
   RUNG wire#powerrail
      Contact( "AlwaysTRUE" )
      I_Contact( "Is_extras_K1" )
      Contact( #set_Motor2 )
      Contact( "Is_loading_K3" )
      I_Contact( "IsRunNetwork_P2" )
      I_Contact( "IsRunNetwork_P3" )
      I_Contact( "IsRunNetwork_P4" )
      Contact( "IsRunNetwork_P1" )
      S_Coil( "Is_extras_K1_P1" )
   END_RUNG
   // the same network as SCL:
   IF "AlwaysTRUE" AND NOT "Is_extras_K1" AND #set_Motor2 AND "Is_loading_K3" AND NOT "IsRunNetwork_P2" AND NOT "IsRunNetwork_P3" AND NOT "IsRunNetwork_P4" AND "IsRunNetwork_P1" THEN
       "Is_extras_K1_P1" := TRUE;
   END_IF;
END_REGION

REGION Network 11: Znacznik motor P2 dodatkowy nr 1
   RUNG wire#powerrail
      Contact( "AlwaysTRUE" )
      I_Contact( "Is_extras_K1" )
      Contact( #set_Motor2 )
      Contact( "Is_loading_K3" )
      I_Contact( "IsRunNetwork_P1" )
      I_Contact( "IsRunNetwork_P3" )
      I_Contact( "IsRunNetwork_P4" )
      Contact( "IsRunNetwork_P2" )
      S_Coil( "Is_extras_K1_P2" )
   END_RUNG
   // the same network as SCL:
   IF "AlwaysTRUE" AND NOT "Is_extras_K1" AND #set_Motor2 AND "Is_loading_K3" AND NOT "IsRunNetwork_P1" AND NOT "IsRunNetwork_P3" AND NOT "IsRunNetwork_P4" AND "IsRunNetwork_P2" THEN
       "Is_extras_K1_P2" := TRUE;
   END_IF;
END_REGION

REGION Network 12: Znacznik motor P3 dodatkowy nr 1
   RUNG wire#powerrail
      Contact( "AlwaysTRUE" )
      I_Contact( "Is_extras_K1" )
      Contact( #set_Motor2 )
      Contact( "Is_loading_K3" )
      I_Contact( "IsRunNetwork_P1" )
      I_Contact( "IsRunNetwork_P2" )
      I_Contact( "IsRunNetwork_P4" )
      Contact( "IsRunNetwork_P3" )
      S_Coil( "Is_extras_K1_P3" )
   END_RUNG
   // the same network as SCL:
   IF "AlwaysTRUE" AND NOT "Is_extras_K1" AND #set_Motor2 AND "Is_loading_K3" AND NOT "IsRunNetwork_P1" AND NOT "IsRunNetwork_P2" AND NOT "IsRunNetwork_P4" AND "IsRunNetwork_P3" THEN
       "Is_extras_K1_P3" := TRUE;
   END_IF;
END_REGION

REGION Network 13: Znacznik motor P3 dodatkowy nr 1 / Znacznik motor P4 dodatkowy nr 1
   RUNG wire#powerrail
      Contact( "AlwaysTRUE" )
      I_Contact( "Is_extras_K1" )
      Contact( #set_Motor2 )
      Contact( "Is_loading_K3" )
      I_Contact( "IsRunNetwork_P1" )
      I_Contact( "IsRunNetwork_P2" )
      I_Contact( "IsRunNetwork_P3" )
      Contact( "IsRunNetwork_P4" )
      S_Coil( "Is_extras_K1_P4" )
   END_RUNG
   // the same network as SCL:
   IF "AlwaysTRUE" AND NOT "Is_extras_K1" AND #set_Motor2 AND "Is_loading_K3" AND NOT "IsRunNetwork_P1" AND NOT "IsRunNetwork_P2" AND NOT "IsRunNetwork_P3" AND "IsRunNetwork_P4" THEN
       "Is_extras_K1_P4" := TRUE;
   END_IF;
END_REGION

REGION Network 14: Znacznik dodatkowa 1
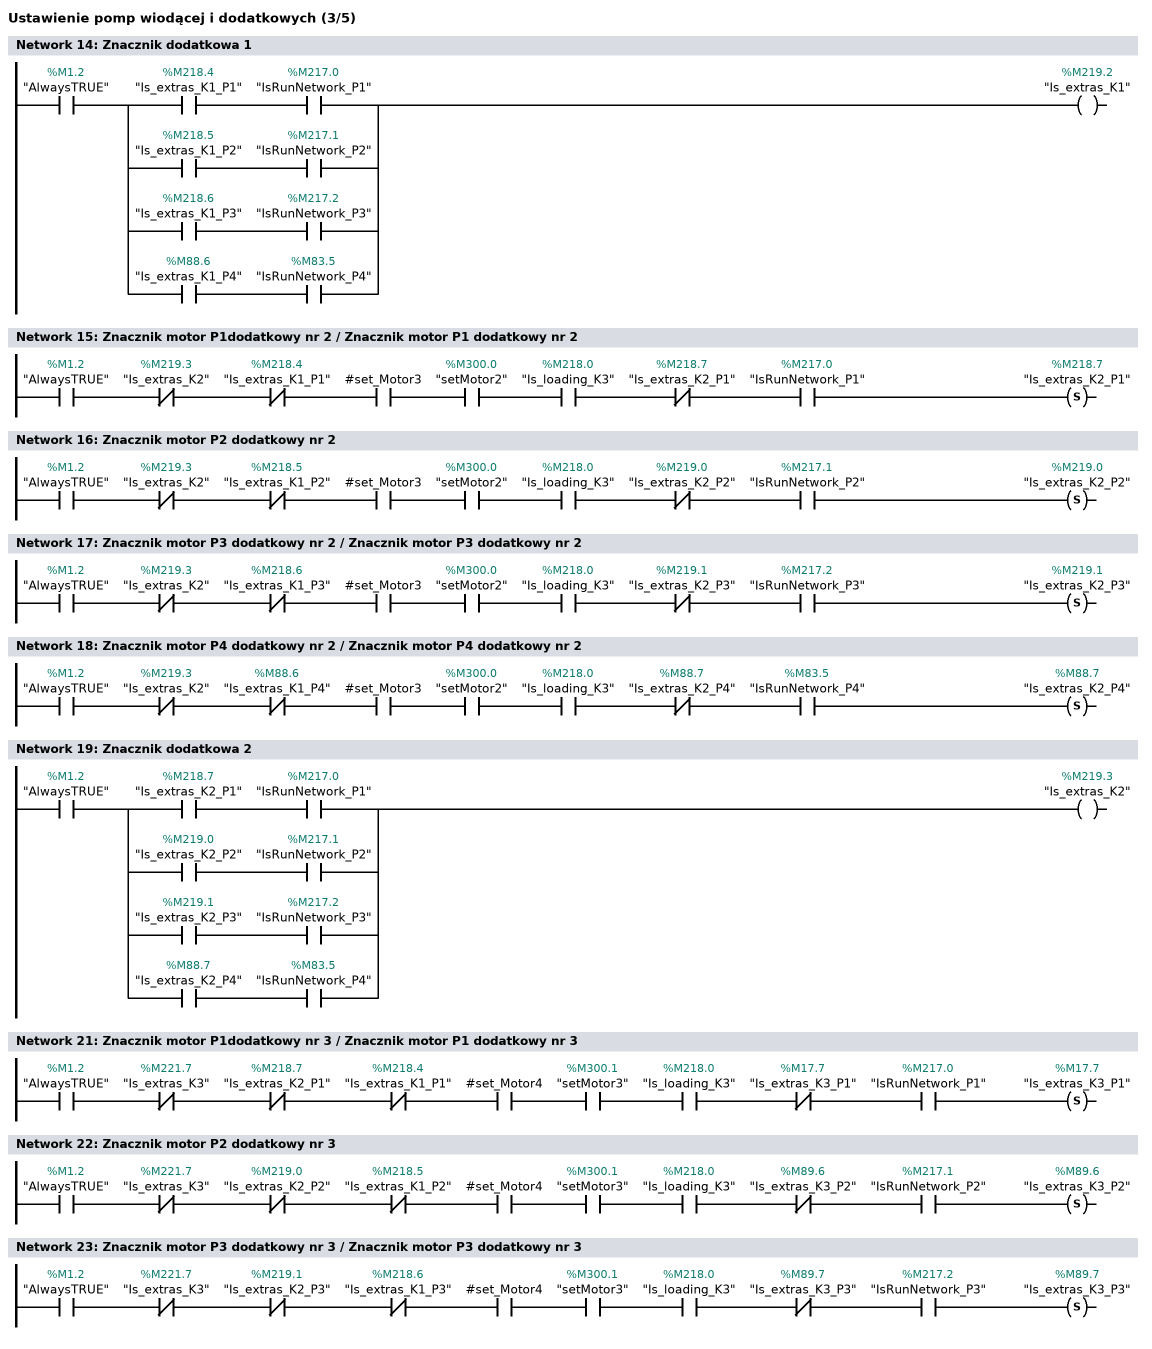
   RUNG wire#powerrail
      Contact( "AlwaysTRUE" )
      wire#w1
      Contact( "Is_extras_K1_P1" )
      Contact( "IsRunNetwork_P1" )
      wire#w2
      Coil( "Is_extras_K1" )
   END_RUNG
   RUNG wire#w1
      Contact( "Is_extras_K1_P2" )
      Contact( "IsRunNetwork_P2" )
   END_RUNG wire#w2
   RUNG wire#w1
      Contact( "Is_extras_K1_P3" )
      Contact( "IsRunNetwork_P3" )
   END_RUNG wire#w2
   RUNG wire#w1
      Contact( "Is_extras_K1_P4" )
      Contact( "IsRunNetwork_P4" )
   END_RUNG wire#w2
   // the same network as SCL:
   "Is_extras_K1" := "AlwaysTRUE" AND (("Is_extras_K1_P1" AND "IsRunNetwork_P1") OR ("Is_extras_K1_P2" AND "IsRunNetwork_P2") OR ("Is_extras_K1_P3" AND "IsRunNetwork_P3") OR ("Is_extras_K1_P4" AND "IsRunNetwork_P4"));
END_REGION

REGION Network 15: Znacznik motor P1dodatkowy nr 2 / Znacznik motor P1 dodatkowy nr 2
   RUNG wire#powerrail
      Contact( "AlwaysTRUE" )
      I_Contact( "Is_extras_K2" )
      I_Contact( "Is_extras_K1_P1" )
      Contact( #set_Motor3 )
      Contact( "setMotor2" )
      Contact( "Is_loading_K3" )
      I_Contact( "Is_extras_K2_P1" )
      Contact( "IsRunNetwork_P1" )
      S_Coil( "Is_extras_K2_P1" )
   END_RUNG
   // the same network as SCL:
   IF "AlwaysTRUE" AND NOT "Is_extras_K2" AND NOT "Is_extras_K1_P1" AND #set_Motor3 AND "setMotor2" AND "Is_loading_K3" AND NOT "Is_extras_K2_P1" AND "IsRunNetwork_P1" THEN
       "Is_extras_K2_P1" := TRUE;
   END_IF;
END_REGION

REGION Network 16: Znacznik motor P2 dodatkowy nr 2
   RUNG wire#powerrail
      Contact( "AlwaysTRUE" )
      I_Contact( "Is_extras_K2" )
      I_Contact( "Is_extras_K1_P2" )
      Contact( #set_Motor3 )
      Contact( "setMotor2" )
      Contact( "Is_loading_K3" )
      I_Contact( "Is_extras_K2_P2" )
      Contact( "IsRunNetwork_P2" )
      S_Coil( "Is_extras_K2_P2" )
   END_RUNG
   // the same network as SCL:
   IF "AlwaysTRUE" AND NOT "Is_extras_K2" AND NOT "Is_extras_K1_P2" AND #set_Motor3 AND "setMotor2" AND "Is_loading_K3" AND NOT "Is_extras_K2_P2" AND "IsRunNetwork_P2" THEN
       "Is_extras_K2_P2" := TRUE;
   END_IF;
END_REGION

REGION Network 17: Znacznik motor P3 dodatkowy nr 2 / Znacznik motor P3 dodatkowy nr 2
   RUNG wire#powerrail
      Contact( "AlwaysTRUE" )
      I_Contact( "Is_extras_K2" )
      I_Contact( "Is_extras_K1_P3" )
      Contact( #set_Motor3 )
      Contact( "setMotor2" )
      Contact( "Is_loading_K3" )
      I_Contact( "Is_extras_K2_P3" )
      Contact( "IsRunNetwork_P3" )
      S_Coil( "Is_extras_K2_P3" )
   END_RUNG
   // the same network as SCL:
   IF "AlwaysTRUE" AND NOT "Is_extras_K2" AND NOT "Is_extras_K1_P3" AND #set_Motor3 AND "setMotor2" AND "Is_loading_K3" AND NOT "Is_extras_K2_P3" AND "IsRunNetwork_P3" THEN
       "Is_extras_K2_P3" := TRUE;
   END_IF;
END_REGION

REGION Network 18: Znacznik motor P4 dodatkowy nr 2 / Znacznik motor P4 dodatkowy nr 2
   RUNG wire#powerrail
      Contact( "AlwaysTRUE" )
      I_Contact( "Is_extras_K2" )
      I_Contact( "Is_extras_K1_P4" )
      Contact( #set_Motor3 )
      Contact( "setMotor2" )
      Contact( "Is_loading_K3" )
      I_Contact( "Is_extras_K2_P4" )
      Contact( "IsRunNetwork_P4" )
      S_Coil( "Is_extras_K2_P4" )
   END_RUNG
   // the same network as SCL:
   IF "AlwaysTRUE" AND NOT "Is_extras_K2" AND NOT "Is_extras_K1_P4" AND #set_Motor3 AND "setMotor2" AND "Is_loading_K3" AND NOT "Is_extras_K2_P4" AND "IsRunNetwork_P4" THEN
       "Is_extras_K2_P4" := TRUE;
   END_IF;
END_REGION

REGION Network 19: Znacznik dodatkowa 2
   RUNG wire#powerrail
      Contact( "AlwaysTRUE" )
      wire#w1
      Contact( "Is_extras_K2_P1" )
      Contact( "IsRunNetwork_P1" )
      wire#w2
      Coil( "Is_extras_K2" )
   END_RUNG
   RUNG wire#w1
      Contact( "Is_extras_K2_P2" )
      Contact( "IsRunNetwork_P2" )
   END_RUNG wire#w2
   RUNG wire#w1
      Contact( "Is_extras_K2_P3" )
      Contact( "IsRunNetwork_P3" )
   END_RUNG wire#w2
   RUNG wire#w1
      Contact( "Is_extras_K2_P4" )
      Contact( "IsRunNetwork_P4" )
   END_RUNG wire#w2
   // the same network as SCL:
   "Is_extras_K2" := "AlwaysTRUE" AND (("Is_extras_K2_P1" AND "IsRunNetwork_P1") OR ("Is_extras_K2_P2" AND "IsRunNetwork_P2") OR ("Is_extras_K2_P3" AND "IsRunNetwork_P3") OR ("Is_extras_K2_P4" AND "IsRunNetwork_P4"));
END_REGION

REGION Network 21: Znacznik motor P1dodatkowy nr 3 / Znacznik motor P1 dodatkowy nr 3
   RUNG wire#powerrail
      Contact( "AlwaysTRUE" )
      I_Contact( "Is_extras_K3" )
      I_Contact( "Is_extras_K2_P1" )
      I_Contact( "Is_extras_K1_P1" )
      Contact( #set_Motor4 )
      Contact( "setMotor3" )
      Contact( "Is_loading_K3" )
      I_Contact( "Is_extras_K3_P1" )
      Contact( "IsRunNetwork_P1" )
      S_Coil( "Is_extras_K3_P1" )
   END_RUNG
   // the same network as SCL:
   IF "AlwaysTRUE" AND NOT "Is_extras_K3" AND NOT "Is_extras_K2_P1" AND NOT "Is_extras_K1_P1" AND #set_Motor4 AND "setMotor3" AND "Is_loading_K3" AND NOT "Is_extras_K3_P1" AND "IsRunNetwork_P1" THEN
       "Is_extras_K3_P1" := TRUE;
   END_IF;
END_REGION

REGION Network 22: Znacznik motor P2 dodatkowy nr 3
   RUNG wire#powerrail
      Contact( "AlwaysTRUE" )
      I_Contact( "Is_extras_K3" )
      I_Contact( "Is_extras_K2_P2" )
      I_Contact( "Is_extras_K1_P2" )
      Contact( #set_Motor4 )
      Contact( "setMotor3" )
      Contact( "Is_loading_K3" )
      I_Contact( "Is_extras_K3_P2" )
      Contact( "IsRunNetwork_P2" )
      S_Coil( "Is_extras_K3_P2" )
   END_RUNG
   // the same network as SCL:
   IF "AlwaysTRUE" AND NOT "Is_extras_K3" AND NOT "Is_extras_K2_P2" AND NOT "Is_extras_K1_P2" AND #set_Motor4 AND "setMotor3" AND "Is_loading_K3" AND NOT "Is_extras_K3_P2" AND "IsRunNetwork_P2" THEN
       "Is_extras_K3_P2" := TRUE;
   END_IF;
END_REGION

REGION Network 23: Znacznik motor P3 dodatkowy nr 3 / Znacznik motor P3 dodatkowy nr 3
   RUNG wire#powerrail
      Contact( "AlwaysTRUE" )
      I_Contact( "Is_extras_K3" )
      I_Contact( "Is_extras_K2_P3" )
      I_Contact( "Is_extras_K1_P3" )
      Contact( #set_Motor4 )
      Contact( "setMotor3" )
      Contact( "Is_loading_K3" )
      I_Contact( "Is_extras_K3_P3" )
      Contact( "IsRunNetwork_P3" )
      S_Coil( "Is_extras_K3_P3" )
   END_RUNG
   // the same network as SCL:
   IF "AlwaysTRUE" AND NOT "Is_extras_K3" AND NOT "Is_extras_K2_P3" AND NOT "Is_extras_K1_P3" AND #set_Motor4 AND "setMotor3" AND "Is_loading_K3" AND NOT "Is_extras_K3_P3" AND "IsRunNetwork_P3" THEN
       "Is_extras_K3_P3" := TRUE;
   END_IF;
END_REGION

REGION Network 24: Znacznik motor P4 dodatkowy nr 3
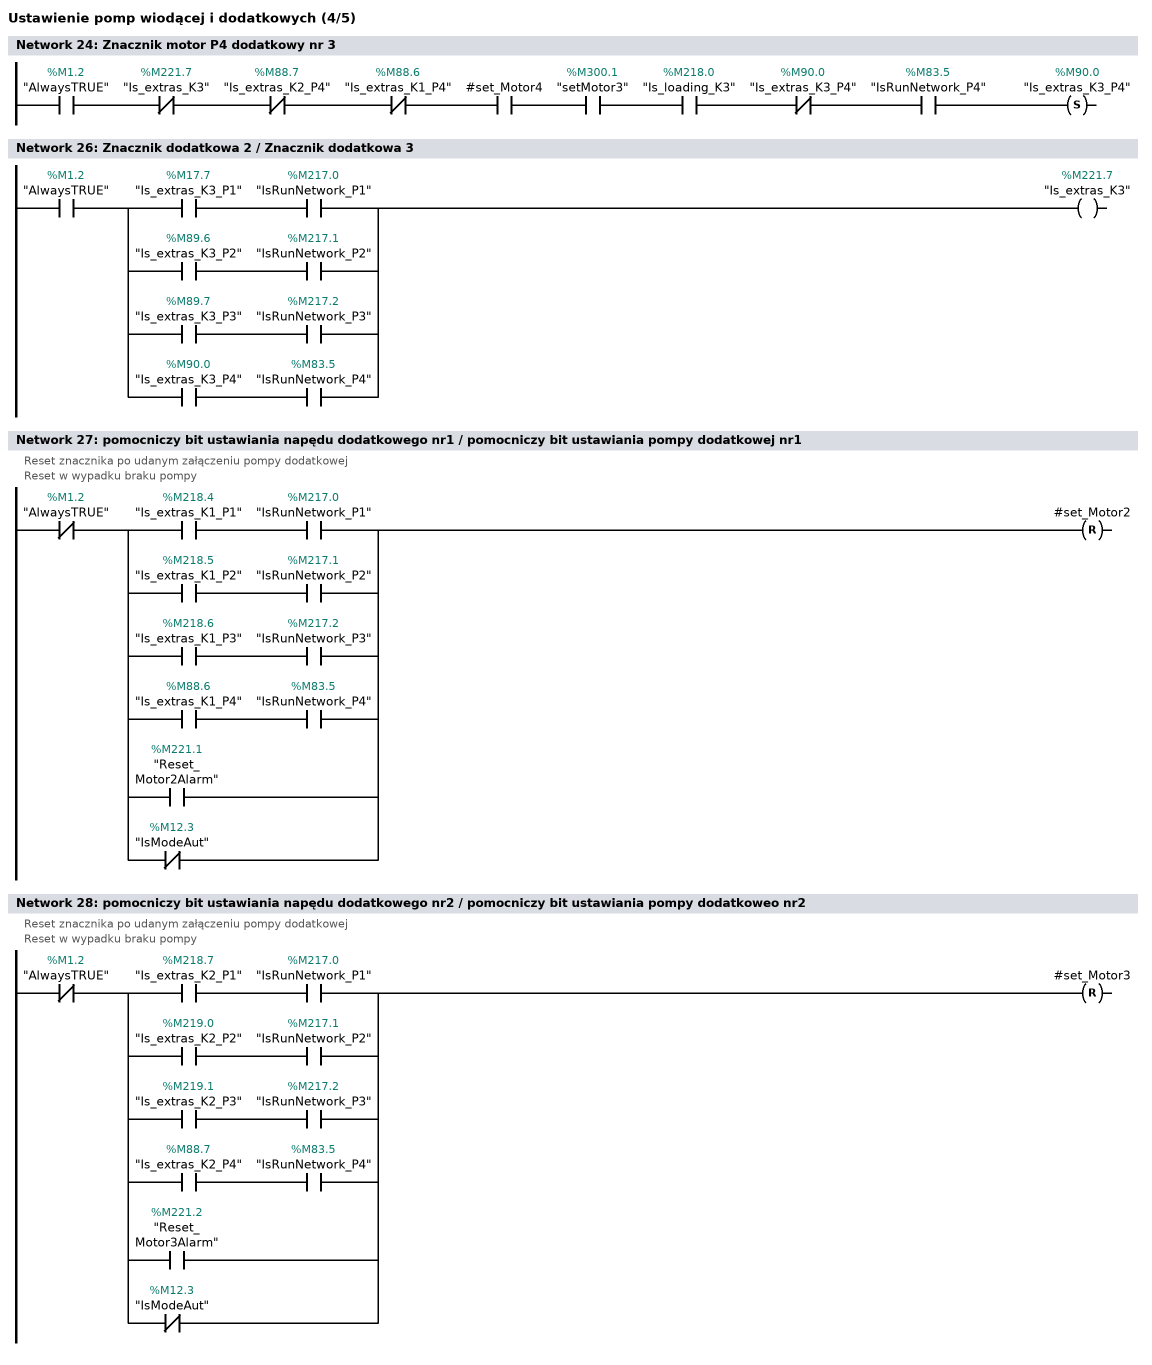
   RUNG wire#powerrail
      Contact( "AlwaysTRUE" )
      I_Contact( "Is_extras_K3" )
      I_Contact( "Is_extras_K2_P4" )
      I_Contact( "Is_extras_K1_P4" )
      Contact( #set_Motor4 )
      Contact( "setMotor3" )
      Contact( "Is_loading_K3" )
      I_Contact( "Is_extras_K3_P4" )
      Contact( "IsRunNetwork_P4" )
      S_Coil( "Is_extras_K3_P4" )
   END_RUNG
   // the same network as SCL:
   IF "AlwaysTRUE" AND NOT "Is_extras_K3" AND NOT "Is_extras_K2_P4" AND NOT "Is_extras_K1_P4" AND #set_Motor4 AND "setMotor3" AND "Is_loading_K3" AND NOT "Is_extras_K3_P4" AND "IsRunNetwork_P4" THEN
       "Is_extras_K3_P4" := TRUE;
   END_IF;
END_REGION

REGION Network 26: Znacznik dodatkowa 2 / Znacznik dodatkowa 3
   RUNG wire#powerrail
      Contact( "AlwaysTRUE" )
      wire#w1
      Contact( "Is_extras_K3_P1" )
      Contact( "IsRunNetwork_P1" )
      wire#w2
      Coil( "Is_extras_K3" )
   END_RUNG
   RUNG wire#w1
      Contact( "Is_extras_K3_P2" )
      Contact( "IsRunNetwork_P2" )
   END_RUNG wire#w2
   RUNG wire#w1
      Contact( "Is_extras_K3_P3" )
      Contact( "IsRunNetwork_P3" )
   END_RUNG wire#w2
   RUNG wire#w1
      Contact( "Is_extras_K3_P4" )
      Contact( "IsRunNetwork_P4" )
   END_RUNG wire#w2
   // the same network as SCL:
   "Is_extras_K3" := "AlwaysTRUE" AND (("Is_extras_K3_P1" AND "IsRunNetwork_P1") OR ("Is_extras_K3_P2" AND "IsRunNetwork_P2") OR ("Is_extras_K3_P3" AND "IsRunNetwork_P3") OR ("Is_extras_K3_P4" AND "IsRunNetwork_P4"));
END_REGION

REGION Network 27: pomocniczy bit ustawiania napędu dodatkowego nr1 / pomocniczy bit ustawiania pompy dodatkowej nr1
   // Reset znacznika po udanym załączeniu pompy dodatkowej
   // Reset w wypadku braku pompy
   RUNG wire#powerrail
      I_Contact( "AlwaysTRUE" )
      wire#w1
      Contact( "Is_extras_K1_P1" )
      Contact( "IsRunNetwork_P1" )
      wire#w2
      R_Coil( #set_Motor2 )
   END_RUNG
   RUNG wire#w1
      Contact( "Is_extras_K1_P2" )
      Contact( "IsRunNetwork_P2" )
   END_RUNG wire#w2
   RUNG wire#w1
      Contact( "Is_extras_K1_P3" )
      Contact( "IsRunNetwork_P3" )
   END_RUNG wire#w2
   RUNG wire#w1
      Contact( "Is_extras_K1_P4" )
      Contact( "IsRunNetwork_P4" )
   END_RUNG wire#w2
   RUNG wire#w1
      Contact( "Reset_Motor2Alarm" )
   END_RUNG wire#w2
   RUNG wire#w1
      I_Contact( "IsModeAut" )
   END_RUNG wire#w2
   // the same network as SCL:
   IF NOT "AlwaysTRUE" AND (("Is_extras_K1_P1" AND "IsRunNetwork_P1") OR ("Is_extras_K1_P2" AND "IsRunNetwork_P2") OR ("Is_extras_K1_P3" AND "IsRunNetwork_P3") OR ("Is_extras_K1_P4" AND "IsRunNetwork_P4") OR "Reset_Motor2Alarm" OR NOT "IsModeAut") THEN
       #set_Motor2 := FALSE;
   END_IF;
END_REGION

